	b := UDINT_TO_INT(SIZE) - 1;
	FOR a := 0 TO b DO
		d := d + 1;
		e := e + sbox[d];
		v := sbox[d];
		sbox[d] := sbox[e];
		sbox[e] := v;
		v := sbox[d] + sbox[e];
		BUF[a] :=BUF[a] XOR sbox[v];
	END_FOR;

	POS := POS + SIZE;
	SIZE := MIN(64,end - POS);

	IF SIZE = 0 THEN
		MODE := 3;
	END_IF;
END_CASE;

(* revision history

ks	9. Jan. 2010 rev 1.0
	original version

*)

END_FUNCTION_BLOCK

// POUs/DEMO/SHA1_MD5_DEMO
PROGRAM SHA1_MD5_DEMO
VAR
	text: STRING(OSCAT_BASIC.STRING_LENGTH) := '<4036.1076324381@guildenstern.zeitform.de>';
	MD5_STR : MD5_STR;
	SHA1_STR : SHA1_STR;
	md5_hash : ARRAY [0..15] OF BYTE;
	sha1_hash : ARRAY [0..19] OF BYTE;
	start1 : BOOL := TRUE;
	start2 : BOOL := TRUE;
	done1 : BOOL;
	done2 : BOOL;
	md5_strh : STRING(32);
	sha1_strh : STRING(40);
END_VAR

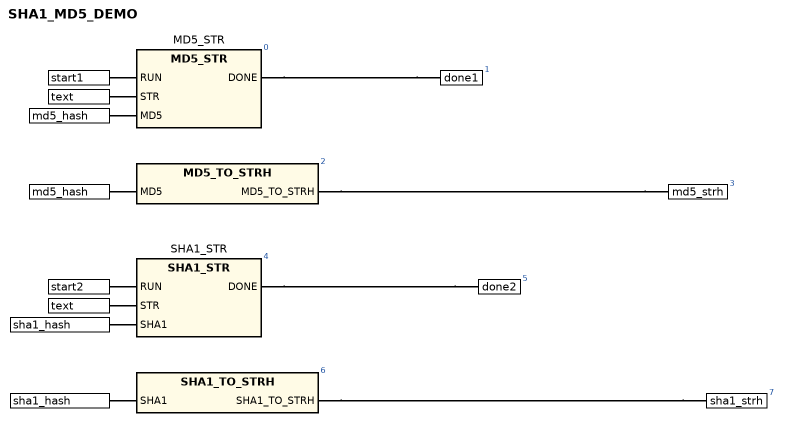
MD5_STR(RUN := start1, STR := text, MD5 := md5_hash);
done1 := MD5_STR.DONE;
md5_strh := MD5_TO_STRH(MD5 := md5_hash);
SHA1_STR(RUN := start2, STR := text, SHA1 := sha1_hash);
done2 := SHA1_STR.DONE;
sha1_strh := SHA1_TO_STRH(SHA1 := sha1_hash);

END_PROGRAM

// POUs/CONVERT/SHA1_STR
FUNCTION_BLOCK SHA1_STR
VAR_INPUT
	RUN: BOOL;
END_VAR
VAR_OUTPUT
	DONE: BOOL;
END_VAR
VAR_IN_OUT
	STR: STRING(OSCAT_BASIC.STRING_LENGTH);
	SHA1 : ARRAY [0..19] OF BYTE;
END_VAR

VAR
	run_last: BOOL;
	SHA1_STREAM : SHA1_STREAM;
	buf : ARRAY [0..63] OF BYTE;
	mode : INT;
	size : UDINT;
	pos : UDINT;
END_VAR

(*
version 1.0	06. dec. 2009
programmer 	ks
tested BY	ks

SHA1_STR berechnet den MD5 Hash eines Strings
*)

CASE mode OF
0:	(* Wait für Start *)
	IF RUN AND NOT run_last THEN
		DONE := FALSE;
		mode := 1; (* Initialisierung *)
		size := LEN(STR);
	END_IF;

2:	(* Data copy and Calc *)
	IF size > 0 THEN
		OSCAT_BASIC._STRING_TO_BUFFER(STR:=MID(STR, UDINT_TO_INT(SIZE), UDINT_TO_INT(POS) + 1), POS:=0, PT:=ADR(buf), SIZE:=SIZEOF(buf));
	END_IF;

3:	DONE := TRUE;
	mode := 0; (* Stop *)

END_CASE;

IF mode > 0 THEN
	SHA1_STREAM(SIZE:=size, MODE:=mode, BUF:=buf, SHA1:=SHA1, POS=>pos);
END_IF;

run_last := RUN;

(* revision history

ks	6. dec. 2009 rev 1.0
	original version

*)

END_FUNCTION_BLOCK

// POUs/CONVERT/SHA1_TO_STRH
FUNCTION SHA1_TO_STRH : STRING(40)
VAR_INPUT
	SHA1 : ARRAY [0..19] OF BYTE;
END_VAR
VAR
	i : INT;
	tmp : BYTE;
	pt : POINTER TO BYTE;
END_VAR
(*
version 1.1	03. dec. 2011
programmer 	ks
tested BY	ks

SHA1_TO_STRH konvertiert das SHA1 Hash Array in einen HEX-String
*)

pt := ADR(SHA1_TO_STRH); (* read output adress to pointer *)

FOR i := 0 TO 19 DO; (* write the 10 hex characters backwards *)
	tmp := SHR(SHA1[i],4);
	PT^ := tmp + SEL(tmp <= 9,87,48);
	pt := pt + 1; (* decrement the pointer *)
	tmp := SHA1[i] AND 2#1111;
	PT^ := tmp + SEL(tmp <= 9,87,48);
	pt := pt + 1; (* decrement the pointer *)
END_FOR;
pt^:= 0; (* write the closing byte for the string *)

(* revision history

ks	6. dec. 2009 rev 1.0
	original version

ks	3. dec. 2011 rev 1.1
	incorrect string size
*)

END_FUNCTION

// POUs/DEMO/SMTP_CLIENT_DEMO
PROGRAM SMTP_CLIENT_DEMO
VAR
(*
	smtp_server: STRING := 'oscat_test%freenet.de:oscat123456@mx.freenet.de';
	smtp_mailfrom: STRING := 'oscat_test@freenet.de';
*)

	SMTP_CLIENT: SMTP_CLIENT;
	smtp_activate: BOOL;
	smtp_timeout: TIME := T#30s;
	smtp_error_t: BYTE;
	smtp_error_c: DWORD;
	smtp_busy: BOOL;
	smtp_done: BOOL;
	smtp_dti: DT;
	smtp_dti_offset: INT := 60;
	smtp_files: STRING(OSCAT_BASIC.STRING_LENGTH) := '';
	smtp_server: STRING := '110876022:oscat123456@mail.gmx.net';
	smtp_mailfrom: STRING := 'oscat@gmx.net;Station_01';
	smtp_mailto: STRING(OSCAT_BASIC.STRING_LENGTH) := 'oscat@gmx.net';
	smtp_subject: STRING := 'Das ist der Betreff';
	smtp_body: STRING(OSCAT_BASIC.STRING_LENGTH) := 'Das ist der Email-Text';
END_VAR
VAR // added by the converter: edge detectors and wires of the graphical bodies
    _w1 : ANY;
END_VAR

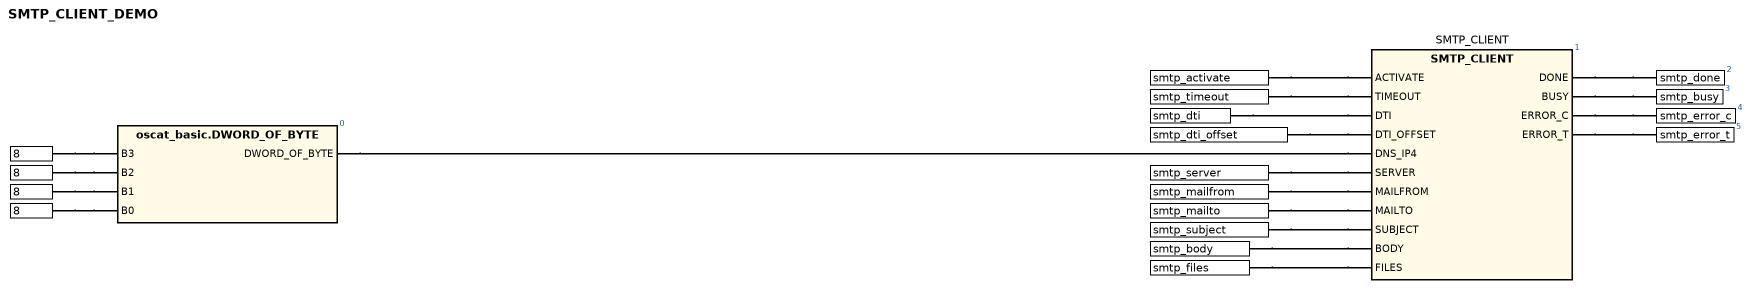
_w1 := oscat_basic.DWORD_OF_BYTE(B3 := 8, B2 := 8, B1 := 8, B0 := 8);
SMTP_CLIENT(
    ACTIVATE := smtp_activate,
    TIMEOUT := smtp_timeout,
    DTI := smtp_dti,
    DTI_OFFSET := smtp_dti_offset,
    DNS_IP4 := _w1,
    SERVER := smtp_server,
    MAILFROM := smtp_mailfrom,
    MAILTO := smtp_mailto,
    SUBJECT := smtp_subject,
    BODY := smtp_body,
    FILES := smtp_files);
smtp_done := SMTP_CLIENT.DONE;
smtp_busy := SMTP_CLIENT.BUSY;
smtp_error_c := SMTP_CLIENT.ERROR_C;
smtp_error_t := SMTP_CLIENT.ERROR_T;

END_PROGRAM

// POUs/NETWORK/SPIDER_ACCESS
FUNCTION_BLOCK SPIDER_ACCESS
VAR_IN_OUT
	IP_C : IP_C;(*IP_Control Verwaltungsstruktur*)
	S_BUF : NETWORK_BUFFER;
	R_BUF : NETWORK_BUFFER;
	VALUE : STRING;
	VAR_NAME : STRING(40);
END_VAR
VAR_INPUT
	MODE : BYTE;
END_VAR
VAR_OUTPUT
	ERROR : DWORD;
END_VAR
VAR
	state : INT;
	st_tmp : STRING(OSCAT_BASIC.STRING_LENGTH);
	URL_DATA : url;
	HTTP_GET : HTTP_GET;
	value_len :	UINT;
	body_len :	UINT;
	mode_save : BYTE;
END_VAR

(*
version 1.1	12. apr. 2011
programmer 	ks
tested by		ks
*)

CASE state OF

00:
	IF MODE > BYTE#0 AND MODE < BYTE#3 THEN
		MODE_SAVE := MODE; (* Modus speichern *)
		(* wenn kein '.' in Name dann ist es eine globale variable *)
		IF FIND(VAR_NAME,'.') = 0 THEN
			st_tmp := CONCAT('%40GV.',VAR_NAME);
		ELSE
			st_tmp := VAR_NAME;
		END_IF;

		IF MODE_SAVE = BYTE#2 THEN (* 2 = Write *)
			VALUE_LEN := INT_TO_UINT(LEN(VALUE));
			st_tmp := CONCAT(st_tmp,'+');
			st_tmp := CONCAT(st_tmp,VALUE);
			URL_DATA:=STRING_TO_URL(STR:= CONCAT('http://x/dir/cgi-bin/writeVal.exe?',st_tmp),DEFAULT_PROTOCOL:='',DEFAULT_PATH:='');
		ELSE
			URL_DATA:=STRING_TO_URL(STR:= CONCAT('http://x/dir/cgi-bin/readVal.exe?',st_tmp),DEFAULT_PROTOCOL:='',DEFAULT_PATH:='');
		END_IF;

		state := 60;
	END_IF;
60:
	IF HTTP_GET.DONE THEN
		IF MODE_SAVE = BYTE#2 THEN (* Write *)
			BODY_LEN := HTTP_GET.BODY_STOP - HTTP_GET.BODY_START + BOOL_TO_UINT(HTTP_GET.BODY_STOP > UINT#0);
			ERROR := BOOL_TO_DWORD(BODY_LEN <> VALUE_LEN);
		ELSE (* Read *)
			IF HTTP_GET.BODY_START > 0 THEN
				VALUE := OSCAT_BASIC.BUFFER_TO_STRING(PT:=ADR(R_BUF.BUFFER),SIZE:=R_BUF.SIZE,START:=UINT_TO_INT(HTTP_GET.BODY_START),STOP:=UINT_TO_INT(HTTP_GET.BODY_STOP));
			ELSE
				VALUE := '';
			END_IF;
		END_IF;
		STATE   := 100;

	ELSIF (HTTP_GET.ERROR > DWORD#00) THEN
		ERROR := HTTP_GET.ERROR;
		STATE   := 100;
	END_IF;

100:
	(* UNLOCK HTTP DATA *)
	IF HTTP_GET.DONE = FALSE THEN
		STATE := 0;
	END_IF;

END_CASE;

(* HTTP_GET *)
HTTP_GET(	IP_C:=IP_C,
			S_BUF:=S_BUF,
			R_BUF:=R_BUF,
			IP4:=DWORD#00,
			GET:=state=60,
			MODE:=BYTE#0,
			UNLOCK_BUF:=state=100,
			URL_DATA:=URL_DATA
			);

(* revision history
ks	18. mar. 2009	rev 1.0
	original version

ks	12. apr. 2011	rev 1.1
	fehlerkorrektur bei buffer_to_string
*)

END_FUNCTION_BLOCK

// POUs/DEMO/SPIDER_DEMO
PROGRAM SPIDER_DEMO
VAR
	SPIDER_ACCESS: SPIDER_ACCESS;
	IP_CONTROL: IP_CONTROL;
	S_BUF: NETWORK_BUFFER;
	R_BUF: NETWORK_BUFFER;
	MODE: BYTE := 1;
	IP_C: IP_C;
	VALUE: STRING;
	VAR_NAME: STRING(40) := 'RTC_SECONDS';
	ERROR: DWORD;
END_VAR
VAR // added by the converter: edge detectors and wires of the graphical bodies
    _w1 : ANY;
END_VAR

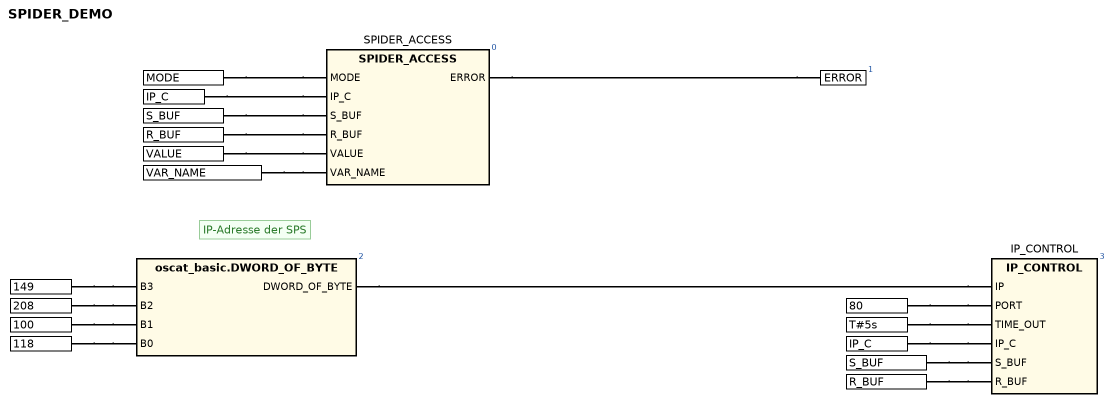
SPIDER_ACCESS(
    MODE := MODE,
    IP_C := IP_C,
    S_BUF := S_BUF,
    R_BUF := R_BUF,
    VALUE := VALUE,
    VAR_NAME := VAR_NAME);
ERROR := SPIDER_ACCESS.ERROR;
// IP-Adresse der SPS
_w1 := oscat_basic.DWORD_OF_BYTE(B3 := 149, B2 := 208, B1 := 100, B0 := 118);
IP_CONTROL(IP := _w1, PORT := 80, TIME_OUT := T#5s, IP_C := IP_C, S_BUF := S_BUF, R_BUF := R_BUF);

END_PROGRAM

// POUs/NETWORK/TELNET_LOG
FUNCTION_BLOCK TELNET_LOG
VAR_IN_OUT
	IP_C : IP_C;
	S_BUF : NETWORK_BUFFER;
	LOG_CL : LOG_CONTROL;
END_VAR
VAR_INPUT
	ENABLE : BOOL;
	OPTION : BYTE := BYTE#2#1000_1100; (* no flush buffer (7) , CR&LF (3), Colors (2), AUTOWRAP (1), Screen-Init (0) *)
	PORT : WORD := 23; (* Port Nummer *)
END_VAR
VAR_OUTPUT
	READY : BOOL;
END_VAR
VAR
	TELNET_PRINT : TELNET_PRINT;
	done : BOOL;
	init : BOOL;
	watchdog : TON;
	ci : INT;
	pi : INT;
	pi_last : INT;
	send : BOOL;
END_VAR

(*
version 1.1	03. Dec. 2011
programmer 	ks
tested BY	ks

TELNET_LOG sendet alle Texte vom LOG_BUFFER an eine TELNET_Konsole
*)

IF NOT init THEN
	init := TRUE;
	IF OPTION > 0 THEN
		TELNET_PRINT.OPTION := OPTION;
	END_IF;
	IF PORT > 0 THEN (* bei portvorgabe wird der standardport überschrieben *)
		TELNET_PRINT.PORT := PORT;
	END_IF;
  	WATCHDOG.PT := T#1ms;
END_IF;

WATCHDOG(IN:=FALSE); (* Timer stoppen *)

ci := LOG_CL.IDX;

(* CONNECT_OFF Flanke auswerten *)
IF IP_C.C_STATE = BYTE#1 THEN
	pi := 0;
	init := FALSE;
END_IF;

REPEAT
	IF pi <> ci AND IP_C.C_STATE > BYTE#127 THEN
		IF pi = 0 AND LOG_CL.RING_MODE THEN pi := ci; END_IF;
		pi_last := pi;
		pi := pi + 1;
		IF pi > LOG_CL.SIZE THEN pi := 1; END_IF;
		SEND := TRUE;
	ELSE
		SEND := FALSE;
	END_IF;

	TELNET_PRINT(	IP_C := IP_C,
					S_BUF := S_BUF,
					ENABLE := ENABLE,
					SEND := SEND,
					TEXT := LOG_CL.MSG[pi],
					BACK_COLOR := DWORD_TO_BYTE(SHL(LOG_CL.MSG_OPTION[pi],8)),
					FRONT_COLOR := DWORD_TO_BYTE(LOG_CL.MSG_OPTION[pi] ));
	READY := TELNET_PRINT.READY;
	done := TELNET_PRINT.DONE;

	IF SEND AND NOT done THEN
		pi := pi_last;
	END_IF;

	WATCHDOG(IN:=TRUE);

UNTIL (WATCHDOG.Q OR NOT done )
END_REPEAT;

(* revision history
ks	14. aug. 2009	rev 1.0
	original version

ks	03. dec. 2011	rev 1.1
	neue parameter und initialisierung optimiert

*)

END_FUNCTION_BLOCK

// POUs/NETWORK/TELNET_PRINT
FUNCTION_BLOCK TELNET_PRINT
VAR_IN_OUT
	IP_C : IP_C;
	S_BUF : NETWORK_BUFFER;
END_VAR
VAR_INPUT
	TEXT : STRING(OSCAT_BASIC.STRING_LENGTH);
	ENABLE : BOOL;
	SEND : BOOL;
	OPTION : BYTE := BYTE#2#1000_1100; (* no flush buffer (7) , CR&LF (3), Colors (2), AUTOWRAP (1), Screen-Init (0) *)
	BACK_COLOR : BYTE;
	FRONT_COLOR : BYTE;
	X_POS : BYTE;
	Y_POS : BYTE;
	PORT : WORD := 23; (* Port Nummer *)
END_VAR
VAR_OUTPUT
	READY : BOOL;
	DONE : BOOL;
END_VAR
VAR
	last_fc : BYTE;
	state : INT;
	x : INT := -1;
	ip_state : BYTE;
	ip_id : BYTE;
	IP_FIFO : IP_FIFO;
	init : BOOL;
	b0_screen_clear : BOOL;
	b1_autowrap : BOOL;
	b2_color : BOOL;
	b3_cr_lr : BOOL;
	b7_no_flush : BOOL;
END_VAR

(*
version 1.4		03. dec. 2011
programmer 		ks
tested by			ks

TELNET_PRINT sendet einem TEXT in Farbe an Position X,Y an eine TELNET-Konsole
*)

READY := IP_C.C_STATE > BYTE#127;
DONE := FALSE;

CASE state OF

00: (* Warten auf Freigabe *)
	IF ENABLE THEN
		state := 10;
		ip_state := BYTE#1; (* Anmelden *)
	END_IF;

10: (* Bei IP_Control anmelden und auf freigabe warten *)
	IF ip_state = BYTE#3 THEN

		(* IP Datenverkehr einrichten *)
		IP_C.C_PORT := PORT; (* Portnummer eintragen *)
		IP_C.C_IP := DWORD#00; (* IP eintragen *)
		IP_C.C_MODE := BYTE#4; (* Mode: TCP+PASSIV+PORT *)
		IP_C.TIME_RESET := TRUE; (* Zeitueberwachung rücksetzen *)
		IP_C.C_ENABLE := TRUE; (* Verbindungsaufbau freigeben *)
		IP_C.R_OBSERVE := FALSE; (* keine Empfangsueberwachung *)
		state := 20;
	END_IF;

20:	IF IP_C.ERROR > DWORD#0 THEN
		IP_C.TIME_RESET := TRUE; (* Fehler rücksetzen *)
	END_IF;
	IF S_BUF.SIZE = UINT#0 THEN (* Datensenden nicht aktiv *)
		IF NOT ENABLE THEN
			ip_state := BYTE#4; (* Verbindung abbauen - Ressource freigeben *)
			IP_C.C_ENABLE := FALSE; (* Verbindungsabbau *)
			state := 0;
		END_IF;
		IF IP_C.C_STATE = BYTE#1 THEN (* positive Flanke Connect off *)
			init := FALSE;
		ELSIF READY THEN (* Verbindung vorhanden *)
			IF IP_C.C_STATE = BYTE#254 AND NOT INIT THEN (* positive Flanke Connect on *)
				(* Var Init ist notwendig, damit der Baustein im selben zyklus mehrmals ausgerufen werden kann *)
				init := TRUE;
				b0_screen_clear := (OPTION AND BYTE#2#0000_0001) > BYTE#0;
				b1_autowrap := (OPTION AND BYTE#2#0000_0010) > BYTE#0;
				b2_color := (OPTION AND BYTE#2#0000_0100) > BYTE#0;
				b3_cr_lr := (OPTION AND BYTE#2#0000_1000) > BYTE#0;
				b7_no_flush := (OPTION AND BYTE#2#1000_0000) > BYTE#0;

				last_fc := NOT FRONT_COLOR; (* aktualisierung der Farben erzwingen !*)
				x := 0;

				(* AUTOWRAP OFF/ON *)
				S_BUF.BUFFER[x] := BYTE#16#1B; (* ESC *)
				x := x +1;
				S_BUF.BUFFER[x] := BYTE#16#5B; (* [ *)
				x := x +1;
				S_BUF.BUFFER[x] := BYTE#16#3F; (* ? *)
				x := x +1;
				S_BUF.BUFFER[x] := BYTE#16#37; (* 7 *)
				x := x +1;
				S_BUF.BUFFER[x] := SEL(b1_autowrap, BYTE#16#6C (* l *),BYTE#16#68 (* h *));

				IF b0_screen_clear THEN
					IF b2_color THEN
						x := x +1;
						S_BUF.BUFFER[x] := BYTE#16#1B; (* ESC *)
						x := x +1;
						S_BUF.BUFFER[x] := BYTE#16#5B; (* [ *)
						x := x +1;
						S_BUF.BUFFER[x] := BYTE#16#30; (* 0 *)
						x := x +1;
						S_BUF.BUFFER[x] := BYTE#16#3B; (* ; *)
						x := x +1;
						S_BUF.BUFFER[x] := BYTE#16#33; (* 3 *)
						x := x +1;
						S_BUF.BUFFER[x] := (FRONT_COLOR AND BYTE#2#00000111) OR BYTE#16#30; (* Einerstelle Farbe Foreground ausgeben *)
						x := x +1;
						S_BUF.BUFFER[x] := BYTE#16#3B; (* ; *)
						x := x +1;
						S_BUF.BUFFER[x] := BYTE#16#34; (* 4 *)
						x := x +1;
						S_BUF.BUFFER[x] := (BACK_COLOR AND BYTE#2#00000111) OR BYTE#16#30; (* Einerstelle Farbe Background ausgeben *)
						x := x +1;
						S_BUF.BUFFER[x] := BYTE#16#6D; (* m *)
					END_IF;
					(* Screen Clear *)
					x := x +1;
					S_BUF.BUFFER[x] := BYTE#16#1B; (* ESC *)
					x := x +1;
					S_BUF.BUFFER[x] := BYTE#16#5B; (* [ *)
					x := x +1;
					S_BUF.BUFFER[x] := BYTE#16#32; (* 2 *)
					x := x +1;
					S_BUF.BUFFER[x] := BYTE#16#4A; (* J *)
				ELSE
					x := x +1;
					S_BUF.BUFFER[x] := BYTE#16#0A; (* neue Zeile *)
				END_IF;
			END_IF;

			(* buffer voll , oder Daten sind vorhanden und kein weiterer Sendewunsch *)
			IF (INT_TO_UINT(x + LEN(TEXT) + 21) > SIZEOF(S_BUF.BUFFER)) OR (x >= 0 AND NOT SEND) THEN
				S_BUF.SIZE := INT_TO_UINT(x + 1); (* Länge eintragen -> Datensenden starten *)
				x := -1;
			ELSIF SEND THEN

				(* aktuelle Farbe bestimmen  *)
				IF b2_color AND FRONT_COLOR <> last_FC THEN
					(* Farbeinstellung: ANSI-Sequenz ESC[X;Y;Zm ausgeben *)
					x := x + 1;
					S_BUF.BUFFER[x] := BYTE#16#1B; (* ESC *)
					x := x + 1;
					S_BUF.BUFFER[x] := BYTE#16#5B; (* [ *)
					(* Farbeinstellung: dunkel oder Hell und blinken bestimmen *)
					IF ((FRONT_COLOR AND BYTE#2#0001_1000) XOR (last_FC AND BYTE#2#0001_1000)) <> BYTE#00 OR TRUE THEN
						x := x + 1;
						S_BUF.BUFFER[x] := BYTE#16#30; (* 0  *)
						x := x + 1;
						S_BUF.BUFFER[x] := BYTE#16#3B; (* ; *)
						(* keine dunklen Farben gewünscht -> dann Bold & Bright *)
						IF (FRONT_COLOR AND BYTE#2#00001000) = BYTE#0 THEN
							(* auf Bold & Bright Farben umstellen *)
							x := x + 1;
							S_BUF.BUFFER[x] := BYTE#16#31; (* 1 *)
							x := x + 1;
							S_BUF.BUFFER[x] := BYTE#16#3B; (* ; *)
						END_IF;
						(* blinkenden Farben gewünscht *)
						IF (FRONT_COLOR AND BYTE#2#00010000) > BYTE#0 THEN
							(* auf Blinkenden Farbe umstellen *)
							x := x + 1;
							S_BUF.BUFFER[x] := BYTE#16#35; (* 5 *)
							x := x + 1;
							S_BUF.BUFFER[x] := BYTE#16#3B; (* ; *)
						END_IF;
					END_IF;
					(* Zehnerstelle Farbe Foreground ausgeben *)
					x := x + 1;
					S_BUF.BUFFER[x] := BYTE#16#33; (* 3 *)
					(* Einerstelle Farbe Foreground ausgeben *)
					x := x + 1;
					S_BUF.BUFFER[x] := (FRONT_COLOR AND BYTE#2#00000111) OR BYTE#16#30;
					x := x + 1;
					S_BUF.BUFFER[x] := BYTE#16#6D; (* m *)
					(* neue Farbe als letzt verwendete speichern *)
					last_FC := FRONT_COLOR;
				END_IF;

				(* Cursor positionieren *)
				IF X_POS > BYTE#0 AND Y_POS > BYTE#0 THEN
					x := x + 1;
					S_BUF.BUFFER[x] := BYTE#16#1B; (* ESC *)
					x := x + 1;
					S_BUF.BUFFER[x] := BYTE#16#5B; (* [ *)
					(* Zehnerstelle Y_POS ausgeben *)
					x := x + 1;
					S_BUF.BUFFER[x] := SHR(OSCAT_BASIC.INT_TO_BCDC(BYTE_TO_INT(Y_POS)),4) OR BYTE#16#30;
					(* Einerstelle Y_POS ausgeben *)
					x := x + 1;
					S_BUF.BUFFER[x] := (OSCAT_BASIC.INT_TO_BCDC(BYTE_TO_INT(Y_POS)) AND BYTE#16#0F) OR BYTE#16#30;
					x := x + 1;
					S_BUF.BUFFER[x] := BYTE#16#3B; (* ; *)
					(* Zehnerstelle X_POS ausgeben *)
					x := x + 1;
					S_BUF.BUFFER[x] := SHR(OSCAT_BASIC.INT_TO_BCDC(BYTE_TO_INT(X_POS)),4) OR BYTE#16#30;
					(* Einerstelle X_POS ausgeben *)
					x := x + 1;
					S_BUF.BUFFER[x] := (OSCAT_BASIC.INT_TO_BCDC(BYTE_TO_INT(X_POS)) AND BYTE#16#0F) OR BYTE#16#30;
					x := x + 1;
					S_BUF.BUFFER[x] := BYTE#16#48; (* H *)
				END_IF;

				(* text ausgeben *)
				IF LEN(TEXT) > 0 THEN
					OSCAT_BASIC._STRING_TO_BUFFER(str:=TEXT,pos:=x + 1,pt :=ADR(S_BUF.BUFFER), size:=SIZEOF(S_BUF.BUFFER));
					x := x + LEN(TEXT);
				END_IF;

				IF b3_cr_lr THEN (* Option: CR,LF ausgeben *)
					x := x + 1;
					S_BUF.BUFFER[x] := BYTE#16#0D;
					x := x + 1;
					S_BUF.BUFFER[x] := BYTE#16#0A;
				END_IF;

				DONE := TRUE; (* Fertig in Buffer eingetragen *)

				IF b7_no_flush THEN (* Option: no buffer flush *)
					(* buffer sofort senden - aktuellen Schreibindex speichern -> Senden anstossen *)
					S_BUF.SIZE := INT_TO_UINT(x + 1);
					x := -1;
				END_IF;
			END_IF;
		END_IF;
	END_IF;
END_CASE;

(* IP_FIFO *)
IP_FIFO(FIFO:=IP_C.FIFO,STATE:=ip_state,ID:=ip_id);

(* revision history
ks	05. jan. 2009	rev 1.0
	original version

ks	20. oct. 2009	rev 1.1
	Networkbuffer und Buffer-funktionen auf Basis 0

ks	20. oct. 2009	rev 1.2
	STRING(OSCAT_BASIC.STRING_LENGTH)

ks	17. may. 2011	rev 1.3
	automatischer re-connect

ks	03. dec. 2011	rev 1.4
	initialisierung verbessert, Port Nummer als Parmeter

*)

END_FUNCTION_BLOCK

// POUs/DEMO/TELNET_LOG_DEMO
PROGRAM TELNET_LOG_DEMO
VAR
	TELNET_LOG: TELNET_LOG;
	IPC: IP_C;
	S_BUF: NETWORK_BUFFER;
	R_BUF: NETWORK_BUFFER;
	READY: BOOL;
	IP_CONTROL: IP_CONTROL;
	TON_1: TON;
	LOG_MSG: LOG_MSG;
END_VAR

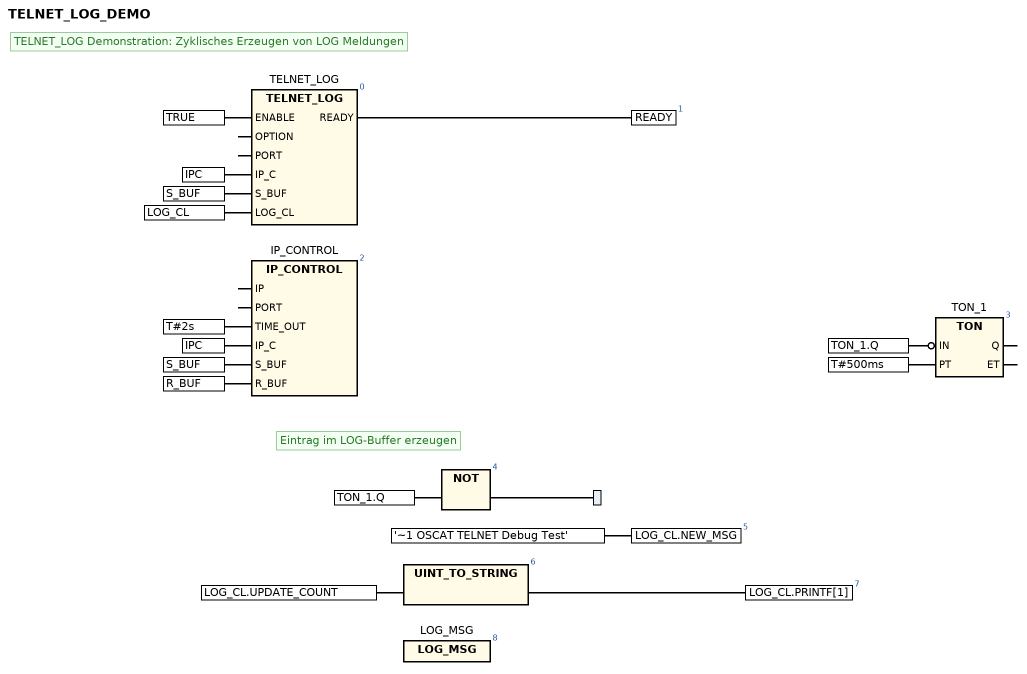
// TELNET_LOG Demonstration: Zyklisches Erzeugen von LOG Meldungen
TELNET_LOG(ENABLE := TRUE, IP_C := IPC, S_BUF := S_BUF, LOG_CL := LOG_CL);
READY := TELNET_LOG.READY;
IP_CONTROL(TIME_OUT := T#2s, IP_C := IPC, S_BUF := S_BUF, R_BUF := R_BUF);
TON_1(IN := NOT TON_1.Q, PT := T#500ms); // TON
// Eintrag im LOG-Buffer erzeugen
(* NOT TON_1.Q; result not used *)
LOG_CL.NEW_MSG := '~1 OSCAT TELNET Debug Test';
LOG_CL.PRINTF[1] := UINT_TO_STRING(LOG_CL.UPDATE_COUNT);
LOG_MSG();

END_PROGRAM

// POUs/DEMO/TELNET_PRINT_DEMO
PROGRAM TELNET_PRINT_DEMO
VAR
	COUNT_BR_1: OSCAT_BASIC.COUNT_BR;
	READY: BOOL;
	TON_1: TON;
	TEXT: STRING;
	TEXT_ATTRIBUTE: BYTE;
	GEN_SIN_1: oscat_basic.GEN_SIN;
	X_POS: BYTE;
	Y_POS: BYTE;
	GEN_SIN_2: oscat_basic.GEN_SIN;
	TELNET_PRINT: TELNET_PRINT;
	DONE: BOOL;
	IP_C: IP_C;
	S_BUF: NETWORK_BUFFER;
	IP_CONTROL: IP_CONTROL;
	R_BUF: NETWORK_BUFFER;
END_VAR
VAR // added by the converter: edge detectors and wires of the graphical bodies
    _w1, _w2 : ANY;
END_VAR

TON_1(IN := NOT TON_1.Q, PT := T#100ms); // TON
COUNT_BR_1(IN := BYTE#1, UP := TON_1.Q AND READY, MX := BYTE#31); // oscat_basic.COUNT_BR
TEXT_ATTRIBUTE := COUNT_BR_1.CNT;
GEN_SIN_1(PT := T#5s, AM := 43.0, OS := 22.0); // oscat_basic.GEN_SIN
_w1 := oscat_basic.STAIR(X := GEN_SIN_1.Out, D := 0.0);
X_POS := REAL_TO_BYTE(_w1);
GEN_SIN_2(PT := T#7s, AM := 24.0, OS := 13.0); // oscat_basic.GEN_SIN
_w2 := oscat_basic.STAIR(X := GEN_SIN_2.Out, D := 0.0);
Y_POS := REAL_TO_BYTE(_w2);
TEXT := CONCAT(STR1 := ' OSCAT TELNET_Print - Test: Color: ', STR2 := BYTE_TO_STRING(TEXT_ATTRIBUTE));
TELNET_PRINT(
    TEXT := TEXT,
    ENABLE := TRUE,
    SEND := TON_1.Q,
    OPTION := BYTE#2#0000_0101,
    BACK_COLOR := BYTE#00,
    FRONT_COLOR := TEXT_ATTRIBUTE,
    X_POS := X_POS,
    Y_POS := Y_POS,
    IP_C := IP_C,
    S_BUF := S_BUF);
READY := TELNET_PRINT.READY;
DONE := TELNET_PRINT.DONE;
IP_CONTROL(TIME_OUT := T#2s, IP_C := IP_C, S_BUF := S_BUF, R_BUF := R_BUF);

END_PROGRAM

// POUs/TELNET_VISION/TN_FRAMEWORK
FUNCTION_BLOCK TN_FRAMEWORK
VAR
	FB_IP_CONTROL : IP_CONTROL;
	FB_TN_INPUT_CONTROL : TN_INPUT_CONTROL;
	FB_TN_INPUT_MENU_BAR : TN_INPUT_MENU_BAR;
	FB_TN_RECEIVE :	TN_RECEIVE;
	FB_TN_SEND_ROWS : TN_SEND_ROWS;
	t : TON;
END_VAR
VAR_IN_OUT
	us_TN_INPUT_CONTROL : us_TN_INPUT_CONTROL;
	us_TN_SCREEN : us_TN_SCREEN;
	us_TN_MENU : us_TN_MENU;
	S_BUF : NETWORK_BUFFER;
	R_BUF : NETWORK_BUFFER;
	IP_C : IP_C;
END_VAR
VAR_INPUT
	PORT : WORD;
END_VAR

(*
version 1.1		17. may 2011
programmer		ks
tested by			ks

TN_FRAMEWORK ist ein Grundgerüst zur Nutzung des TELNET VISION Systems, und beinhält alle Laufzeit Komponenten.
*)

(* Initialisierung / Freigeben der Verbindung *)
IF (NOT IP_C.C_ENABLE) THEN

	(* IP Datenverkehr einrichten *)
	IP_C.C_PORT := SEL(PORT=BYTE#0,PORT,WORD#23); (* Portnummer eintragen *)
	IP_C.C_IP := DWORD#00; (* IP eintragen *)
	IP_C.C_MODE := BYTE#4; (* Mode: TCP+PASSIV+PORT *)
	IP_C.TIME_RESET := TRUE; (* Zeitueberwachung rücksetzen *)
	IP_C.C_ENABLE := TRUE; (* Verbindungsaufbau freigeben *)
	IP_C.R_OBSERVE := FALSE; (* keine Empfangsueberwachung *)

END_IF;

t(IN:= IP_C.ERROR > DWORD#0, PT:=T#5s);
IF t.Q THEN
	IP_C.TIME_RESET := TRUE; (* Error Reset *)
END_IF;

(* Telnet-Menu-Bar *)
FB_TN_INPUT_MENU_BAR(
	Xus_TN_MENU := us_TN_MENU,
	Xus_TN_SCREEN := us_TN_SCREEN);

(* Telnet-Input-Control *)
FB_TN_INPUT_CONTROL(
	Xus_TN_SCREEN := us_TN_SCREEN,
	Xus_TN_INPUT_CONTROL := us_TN_INPUT_CONTROL);

(* Telnet-Data-Send Line-Updates *)
FB_TN_SEND_ROWS(
	IP_C :=IP_C,
	S_BUF :=S_BUF,
	Xus_TN_SCREEN :=us_TN_SCREEN,
	S_BUF_SIZE :=SIZEOF(S_BUF.BUFFER));

(* Telnet-Server *)
FB_IP_CONTROL(
	IP_C :=IP_C,
	S_BUF :=S_BUF,
	R_BUF :=R_BUF,
	IP :=DWORD#00,
	PORT :=WORD#00,
	TIME_OUT :=T#2s);

(* Telnet-Data-Receive *)
FB_TN_RECEIVE(
	R_BUF := R_BUF,
	Xus_TN_SCREEN := us_TN_SCREEN);

(* revision history
ks	10. mai. 2010	rev 1.0
	original version

ks	17. may. 2011	rev 1.1
	automatischer re-connect

ks	05. may. 2012	rev 1.2
	neue parameter PORT
*)

END_FUNCTION_BLOCK

// POUs/TELNET_VISION/TN_INPUT_CONTROL
FUNCTION_BLOCK TN_INPUT_CONTROL
VAR_IN_OUT
	Xus_TN_SCREEN : us_TN_SCREEN;
	Xus_TN_INPUT_CONTROL : us_TN_INPUT_CONTROL;
END_VAR
VAR
	FB_TN_INPUT_SELECT_POPUP : TN_INPUT_SELECT_POPUP;
	FB_TN_INPUT_SELECT_TEXT : TN_INPUT_SELECT_TEXT;
	FB_TN_SC_WRITE_C : TN_SC_WRITE_C;
	FB_TN_INPUT_EDIT_LINE : TN_INPUT_EDIT_LINE;
END_VAR
VAR
	in_index : INT;
	in_Scroll_Offset : INT;
	in_Focus_new : INT;
	in_Focus_alt : INT;
	bo_Tool_Tip_Update : BOOL;
END_VAR

(*
version 1.0		10. mai 2010
programmer		ks
tested by		ks

TN_INPUT_CONTROL dient zur verwaltung und grafischen Darstellung der INPUT_CONTROL Elemente
*)

(* Bearbeitung freigegeben ? *)
IF (Xus_TN_INPUT_CONTROL.bo_Enable = FALSE) OR (Xus_TN_SCREEN.bo_Menue_Bar_Dialog = TRUE) THEN
	RETURN;
END_IF;

(* Fokus Reset durchführen *)
IF (Xus_TN_INPUT_CONTROL.bo_Reset_Fokus = TRUE) THEN
	Xus_TN_INPUT_CONTROL.bo_Reset_Fokus := FALSE;

	FOR in_index := INT#01 TO Xus_TN_INPUT_CONTROL.in_Count DO
		Xus_TN_INPUT_CONTROL.usa_TN_INPUT_CONTROL_DATA[in_index].bo_Focus := FALSE;
	END_FOR;

	IF (Xus_TN_INPUT_CONTROL.in_Count >= INT#01) THEN
		Xus_TN_INPUT_CONTROL.usa_TN_INPUT_CONTROL_DATA[1].bo_Focus := TRUE;
		Xus_TN_INPUT_CONTROL.in_Focus_at := INT#01;
	END_IF;

	Xus_TN_INPUT_CONTROL.bo_Update_all := TRUE;
END_IF;

IF (Xus_TN_SCREEN.bo_Modal_Dialog = FALSE) THEN
	(* TAB-Taste für Control-element wechsel auswerten *)
	IF (Xus_TN_SCREEN.by_Input_Exten_Code = BYTE#09) THEN

		in_Scroll_Offset := INT#01;

		(* Cursor-Oben Taste *)
	ELSIF (Xus_TN_SCREEN.by_Input_Exten_Code = BYTE#65) THEN

		in_Scroll_Offset := -1;

		(* Cursor-unten Taste *)
	ELSIF (Xus_TN_SCREEN.by_Input_Exten_Code = BYTE#66) THEN

		in_Scroll_Offset := INT#01;

	END_IF;
END_IF;

IF (in_Scroll_Offset <> INT#00) THEN  
	(* Grenzwerte überprüfen                                            *)

	Xus_TN_INPUT_CONTROL.in_Focus_at:=LIMIT(INT#01,Xus_TN_INPUT_CONTROL.in_Focus_at,Xus_TN_INPUT_CONTROL.in_Count);

	in_Focus_new := Xus_TN_INPUT_CONTROL.in_Focus_at + in_Scroll_Offset;

	IF (in_Focus_new > Xus_TN_INPUT_CONTROL.in_Count) THEN
		in_Focus_new := INT#1;
	END_IF;

	IF (in_Focus_new < INT#01) THEN
		in_Focus_new := Xus_TN_INPUT_CONTROL.in_Count;
	END_IF;

	in_Focus_alt := Xus_TN_INPUT_CONTROL.in_Focus_at;

	(* aktuellen Element den Fokus entziehen *)
	Xus_TN_INPUT_CONTROL.usa_TN_INPUT_CONTROL_DATA[in_Focus_alt].bo_Focus := FALSE;
	Xus_TN_INPUT_CONTROL.usa_TN_INPUT_CONTROL_DATA[in_Focus_alt].bo_Update_Input := TRUE;

	(* neuem Element den Fokus geben *)
	Xus_TN_INPUT_CONTROL.usa_TN_INPUT_CONTROL_DATA[in_Focus_new].bo_Focus  := TRUE;
	Xus_TN_INPUT_CONTROL.usa_TN_INPUT_CONTROL_DATA[in_Focus_new].bo_Update_Input := TRUE;

	Xus_TN_INPUT_CONTROL.in_Focus_at := in_Focus_new;

	bo_Tool_Tip_Update := TRUE;
	in_Scroll_Offset := INT#00;

END_IF;

(* Alle Elemente updaten ? *)
IF (Xus_TN_INPUT_CONTROL.bo_Update_all = TRUE) THEN
	FOR in_index := 1 TO Xus_TN_INPUT_CONTROL.in_Count DO
		Xus_TN_INPUT_CONTROL.usa_TN_INPUT_CONTROL_DATA[in_index].bo_Update_All := TRUE;
	END_FOR;
	Xus_TN_INPUT_CONTROL.bo_Update_all := FALSE;
	bo_Tool_Tip_Update := TRUE;
END_IF;

FOR in_index := 1 TO Xus_TN_INPUT_CONTROL.in_Count DO

	IF (Xus_TN_INPUT_CONTROL.usa_TN_INPUT_CONTROL_DATA[in_index].in_Type > INT#00) THEN

		IF (Xus_TN_INPUT_CONTROL.usa_TN_INPUT_CONTROL_DATA[in_index].bo_Focus = TRUE) THEN

			Xus_TN_INPUT_CONTROL.usa_TN_INPUT_CONTROL_DATA[in_index].by_Input_ASCII_Code  := Xus_TN_SCREEN.by_Input_ASCII_Code;
			Xus_TN_INPUT_CONTROL.usa_TN_INPUT_CONTROL_DATA[in_index].by_Input_Exten_Code  := Xus_TN_SCREEN.by_Input_Exten_Code;
			Xus_TN_INPUT_CONTROL.usa_TN_INPUT_CONTROL_DATA[in_index].bo_Input_ASCII_IsNum := Xus_TN_SCREEN.bo_Input_ASCII_IsNum;

			(* Tool-Tip Text ausgeben *)
			IF (bo_Tool_Tip_Update = TRUE) THEN

				FB_TN_SC_WRITE_C(	Iin_Y := Xus_TN_INPUT_CONTROL.in_ToolTip_Y,
									Iin_X := Xus_TN_INPUT_CONTROL.in_ToolTip_X,
									Iby_ATTR := Xus_TN_INPUT_CONTROL.by_ToolTip_Attr,
									Iin_OPTION := INT#02, (* Center-String *)
									Iin_LENGTH := Xus_TN_INPUT_CONTROL.in_ToolTip_Size,
									Ist_STRING := Xus_TN_INPUT_CONTROL.usa_TN_INPUT_CONTROL_DATA[in_index].st_Input_ToolTip,
									Xus_TN_SCREEN := Xus_TN_SCREEN);

				(* Flag rücksetzen *)
				bo_Tool_Tip_Update := FALSE;
			END_IF;
		END_IF;

		CASE Xus_TN_INPUT_CONTROL.usa_TN_INPUT_CONTROL_DATA[in_index].in_Type OF
		1:
			(* Edit-Line bearbeiten *)
			FB_TN_INPUT_EDIT_LINE(	Xus_TN_INPUT_CONTROL_DATA := Xus_TN_INPUT_CONTROL.usa_TN_INPUT_CONTROL_DATA[in_index],
									Xus_TN_SCREEN := Xus_TN_SCREEN);
		2:
			(* Select-Text bearbeiten *)
			FB_TN_INPUT_SELECT_TEXT(	Xus_TN_INPUT_CONTROL_DATA := Xus_TN_INPUT_CONTROL.usa_TN_INPUT_CONTROL_DATA[in_index],
										Xus_TN_SCREEN := Xus_TN_SCREEN);
		3:
			(* Select-Popup bearbeiten *)
			FB_TN_INPUT_SELECT_POPUP(	Xus_TN_INPUT_CONTROL_DATA := Xus_TN_INPUT_CONTROL.usa_TN_INPUT_CONTROL_DATA[in_index],
										Xus_TN_SCREEN := Xus_TN_SCREEN);
		END_CASE;

		IF (Xus_TN_INPUT_CONTROL.usa_TN_INPUT_CONTROL_DATA[in_index].bo_Focus = TRUE) THEN

			(* Cursor position von Element auf Screen übertragen *)
			Xus_TN_SCREEN.in_Cursor_X := Xus_TN_INPUT_CONTROL.usa_TN_INPUT_CONTROL_DATA[in_index].in_Cursor_X;
			Xus_TN_SCREEN.in_Cursor_Y := Xus_TN_INPUT_CONTROL.usa_TN_INPUT_CONTROL_DATA[in_index].in_Cursor_Y;

		END_IF;
	END_IF;
END_FOR;

(* revision history
ks	10. mai. 2010	rev 1.0
	original version
*)

END_FUNCTION_BLOCK

// POUs/TELNET_VISION/TN_INPUT_SELECT_POPUP
FUNCTION_BLOCK TN_INPUT_SELECT_POPUP
VAR
	in_index : INT;
	in_Element_Count : INT;
	by_Cur_Key : BYTE;
	by_Attr : BYTE;
	st_String : STRING;
END_VAR
VAR
	us_TN_MENU_POPUP : us_TN_MENU_POPUP;
	FB_TN_INPUT_MENU_POPUP : TN_INPUT_MENU_POPUP;
	FB_TN_SC_WRITE : TN_SC_WRITE;
END_VAR
VAR_IN_OUT
	Xus_TN_SCREEN : us_TN_SCREEN;
	Xus_TN_INPUT_CONTROL_DATA : us_TN_INPUT_CONTROL_DATA;
END_VAR

(*
version 1.1		06. apr 2011
programmer		ks
tested by			ks

TN_SELECT_POPUP dient zur verwaltung und darstellung eines POPUP-Dialogs zur Elementeauswahl
*)

(* Benutzereingabe auswerten -> Selektion Text n *)
IF (Xus_TN_INPUT_CONTROL_DATA.bo_Focus = TRUE) THEN

	by_Cur_Key := Xus_TN_INPUT_CONTROL_DATA.by_Input_Exten_Code;

	IF (us_TN_MENU_POPUP.bo_Activ = FALSE) THEN
		us_TN_MENU_POPUP.by_Input_Exten_Code := BYTE#00;

		(* Return-Taste auswerten *)
		IF (by_Cur_Key = BYTE#13) THEN
			(* Popup-Menu parameter übergeben *)
			us_TN_MENU_POPUP.in_Y := Xus_TN_INPUT_CONTROL_DATA.in_Y;
			us_TN_MENU_POPUP.in_X := Xus_TN_INPUT_CONTROL_DATA.in_X;
			us_TN_MENU_POPUP.by_Attr_mF := Xus_TN_INPUT_CONTROL_DATA.by_Attr_mF;
			us_TN_MENU_POPUP.by_Attr_oF := Xus_TN_INPUT_CONTROL_DATA.by_Attr_oF;
			us_TN_MENU_POPUP.st_Menu_Text := Xus_TN_INPUT_CONTROL_DATA.st_Input_Data;
			us_TN_MENU_POPUP.bo_Create := TRUE;
			us_TN_MENU_POPUP.in_Cur_Item := INT#00;
		END_IF;

		IF (us_TN_MENU_POPUP.in_Cur_Item > INT#00) THEN
			Xus_TN_INPUT_CONTROL_DATA.in_selected := us_TN_MENU_POPUP.in_Cur_Item;
			Xus_TN_INPUT_CONTROL_DATA.bo_Input_Entered := TRUE;
			Xus_TN_INPUT_CONTROL_DATA.bo_Update_Input := TRUE;
			us_TN_MENU_POPUP.in_Cur_Item := INT#00;
		END_IF;

	ELSE
		us_TN_MENU_POPUP.by_Input_Exten_Code := by_Cur_Key;
	END_IF;

	(* Popup-Menu zyklisch aufrufen *)
	FB_TN_INPUT_MENU_POPUP(Xus_TN_MENU_POPUP := us_TN_MENU_POPUP, Xus_TN_SCREEN := Xus_TN_SCREEN);

END_IF;

(* Aktualisierung der Anzeige *)
IF (Xus_TN_INPUT_CONTROL_DATA.bo_Update_Input = TRUE) OR (Xus_TN_INPUT_CONTROL_DATA.bo_Update_All = TRUE) THEN

	(* Title-Text ausgeben *)
	IF Xus_TN_INPUT_CONTROL_DATA.bo_Update_All = TRUE THEN

		IF (Xus_TN_INPUT_CONTROL_DATA.in_Title_X_Offset = INT#00) AND (Xus_TN_INPUT_CONTROL_DATA.in_Title_Y_Offset = INT#00) THEN
			(* wenn Offset X,Y =0 dann Titlestring links vom Element positionieren *)
			FB_TN_SC_WRITE.Iin_Y := Xus_TN_INPUT_CONTROL_DATA.in_Y;
			FB_TN_SC_WRITE.Iin_X := Xus_TN_INPUT_CONTROL_DATA.in_X - LEN(Xus_TN_INPUT_CONTROL_DATA.st_Title_String);

		ELSE
			(* Title-Text durch Row, Color-Offset ausgeben *)
			FB_TN_SC_WRITE.Iin_Y := Xus_TN_INPUT_CONTROL_DATA.in_Y + Xus_TN_INPUT_CONTROL_DATA.in_Title_Y_Offset;
			FB_TN_SC_WRITE.Iin_X := Xus_TN_INPUT_CONTROL_DATA.in_X + Xus_TN_INPUT_CONTROL_DATA.in_Title_X_Offset;
		END_IF;

		(* Title-Text durch Row, Color-Offset ausgeben *)
		FB_TN_SC_WRITE(	Iby_ATTR := Xus_TN_INPUT_CONTROL_DATA.by_Title_Attr,
						Ist_STRING := Xus_TN_INPUT_CONTROL_DATA.st_Title_String,
						Xus_TN_SCREEN := Xus_TN_SCREEN);
	END_IF;

	in_Element_Count := ELEMENT_COUNT(SEP:=BYTE#35,ELEMENT:=Xus_TN_INPUT_CONTROL_DATA.st_Input_Data);

	IF in_Element_Count > INT#00 THEN

		Xus_TN_INPUT_CONTROL_DATA.in_selected:=LIMIT(1,Xus_TN_INPUT_CONTROL_DATA.in_selected,in_Element_Count);

		in_index := Xus_TN_INPUT_CONTROL_DATA.in_selected;

		st_String := ELEMENT_GET(SEP:=BYTE#35,POS:=in_index - 1,ELEMENT:=Xus_TN_INPUT_CONTROL_DATA.st_Input_Data);

		st_String:= OSCAT_BASIC.FIX(str:=st_String,
						L:=LEN(Xus_TN_INPUT_CONTROL_DATA.st_Input_Mask),
						C:=BYTE#32,
						M:=Xus_TN_INPUT_CONTROL_DATA.in_Input_Option);


		Xus_TN_INPUT_CONTROL_DATA.st_Input_String := st_String;

		IF Xus_TN_INPUT_CONTROL_DATA.bo_Focus = TRUE THEN
			by_Attr := Xus_TN_INPUT_CONTROL_DATA.by_Attr_mF;
		ELSE
			by_Attr := Xus_TN_INPUT_CONTROL_DATA.by_Attr_oF;
		END_IF;

		FB_TN_SC_WRITE(	Iin_X := Xus_TN_INPUT_CONTROL_DATA.in_X,
								Iin_Y := Xus_TN_INPUT_CONTROL_DATA.in_Y,
								Iby_ATTR := by_Attr,
								Ist_STRING := st_String,
								Xus_TN_SCREEN := Xus_TN_SCREEN );
	END_IF;

	(* Cursor auf aktuelle Position setzen *)
	Xus_TN_INPUT_CONTROL_DATA.in_Cursor_X := Xus_TN_INPUT_CONTROL_DATA.in_X;
	Xus_TN_INPUT_CONTROL_DATA.in_Cursor_Y := Xus_TN_INPUT_CONTROL_DATA.in_Y;

	(* Update-Flag's rücksetzen *)
	Xus_TN_INPUT_CONTROL_DATA.bo_Update_All   := FALSE;
	Xus_TN_INPUT_CONTROL_DATA.bo_Update_Input := FALSE;

END_IF;

(* revision history

ks	06. apr. 2011	rev 1.1
	list_len und list_get durch element_count und element_get ersetzt

ks	10. mai. 2010	rev 1.0
	original version
*)

END_FUNCTION_BLOCK

// POUs/TELNET_VISION/TN_INPUT_MENU_POPUP
FUNCTION_BLOCK TN_INPUT_MENU_POPUP
VAR
	FB_TN_SC_AREA_SAVE : TN_SC_AREA_SAVE;
	FB_TN_SC_AREA_RESTORE : TN_SC_AREA_RESTORE;
	FB_TN_SC_LINE : TN_SC_LINE;
	FB_TN_SC_ADD_SHADOW : TN_SC_ADD_SHADOW;
	FB_TN_SC_BOX : TN_SC_BOX;
	FB_TN_SC_WRITE_C : TN_SC_WRITE_C;
END_VAR
VAR
	in_ROW : INT;
	in_ROWS : INT;
	in_COL : INT;
	in_COLS : INT;
	in_index : INT;
	in_Count : INT;
	in_Scroll_Offset : INT;
	by_ATTR : BYTE;
END_VAR
VAR_IN_OUT
	Xus_TN_MENU_POPUP : us_TN_MENU_POPUP;
	Xus_TN_SCREEN : us_TN_SCREEN;
END_VAR

(*
version 1.1		06. apr 2011
programmer		ks
tested by			ks

TN_MENU_POPUP dient zur verwaltung und darstellung eines MENU-POPUP
*)

(* sicherstellen das rechteck immer innerhalb screen positioniert wird *)

IF (Xus_TN_MENU_POPUP.bo_Activ = FALSE) AND (Xus_TN_MENU_POPUP.bo_Create = TRUE) THEN
	Xus_TN_MENU_POPUP.bo_Activ := TRUE;
	Xus_TN_MENU_POPUP.bo_Create := FALSE;
	Xus_TN_MENU_POPUP.bo_Destroy := FALSE;
	Xus_TN_MENU_POPUP.bo_Update := TRUE;

  (* Sub-Menu-Texte *)

	Xus_TN_MENU_POPUP.in_Menu_E_Count := ELEMENT_COUNT(SEP:=BYTE#35,ELEMENT:=Xus_TN_MENU_POPUP.st_Menu_Text);

	(* Anzahl Zeilen (Sub-Menu-Texte) bestimmen *)
	Xus_TN_MENU_POPUP.in_Rows := Xus_TN_MENU_POPUP.in_Menu_E_Count;

	(* längsten Sub-Menu-Text suchen *)
	Xus_TN_MENU_POPUP.in_Cols := INT#00;

	FOR in_Count := INT#01 TO Xus_TN_MENU_POPUP.in_Rows DO;
		Xus_TN_MENU_POPUP.in_Cols:=MAX(LEN(ELEMENT_GET(SEP:=BYTE#35,POS:=in_Count - 1,ELEMENT:=Xus_TN_MENU_POPUP.st_Menu_Text)),Xus_TN_MENU_POPUP.in_Cols);
	END_FOR;

	(* Horizontale Position überprüfen und korrigieren *)
	IF (Xus_TN_MENU_POPUP.in_X + Xus_TN_MENU_POPUP.in_Cols) > INT#75 THEN
		Xus_TN_MENU_POPUP.in_X := INT#79 - Xus_TN_MENU_POPUP.in_Cols - INT#04;
	END_IF;

  (* Vertikale Position überprüfen und korrigieren *)
	IF (Xus_TN_MENU_POPUP.in_Y + Xus_TN_MENU_POPUP.in_ROWS) > INT#21 THEN
		Xus_TN_MENU_POPUP.in_Y := INT#23 - Xus_TN_MENU_POPUP.in_ROWS - INT#2;
	END_IF;

	Xus_TN_SCREEN.bo_Modal_Dialog := TRUE;

	(* Hintergrund sichern *)
	FB_TN_SC_AREA_SAVE(	Iin_X1 := Xus_TN_MENU_POPUP.in_X,
									Iin_Y1 := Xus_TN_MENU_POPUP.in_Y,
									Iin_X2 := Xus_TN_MENU_POPUP.in_X + Xus_TN_MENU_POPUP.in_Cols + INT#04,
									Iin_Y2 := Xus_TN_MENU_POPUP.in_Y + Xus_TN_MENU_POPUP.in_Rows + INT#02,
									Xus_TN_SCREEN := Xus_TN_SCREEN);

	(* Rahmen für Submenu zeichnen *)
	FB_TN_SC_BOX(	Iin_X1 := Xus_TN_MENU_POPUP.in_X,
					Iin_Y1 := Xus_TN_MENU_POPUP.in_Y,
					Iin_X2 := Xus_TN_MENU_POPUP.in_X + Xus_TN_MENU_POPUP.in_Cols + INT#03,
					Iin_Y2 := Xus_TN_MENU_POPUP.in_Y + Xus_TN_MENU_POPUP.in_Rows + INT#01,
					Iby_FILL := BYTE#32, (* Füllung *)
					Iin_BORDER := INT#01, (* Single-Line Border *)
					Iby_ATTR := Xus_TN_MENU_POPUP.by_Attr_oF,
					Xus_TN_SCREEN := Xus_TN_SCREEN);

	(* Shadow für Submenu zeichnen *)
	FB_TN_SC_ADD_SHADOW(Iin_X1 := Xus_TN_MENU_POPUP.in_X + INT#1,
						Iin_Y1 := Xus_TN_MENU_POPUP.in_Y + INT#1,
						Iin_X2 := Xus_TN_MENU_POPUP.in_X + Xus_TN_MENU_POPUP.in_Cols + INT#04,
						Iin_Y2 := Xus_TN_MENU_POPUP.in_Y + Xus_TN_MENU_POPUP.in_Rows + INT#02,
						Iin_OPTION := INT#00,
						Xus_TN_SCREEN := Xus_TN_SCREEN);

	(* Parameter laden *)
	in_COL := Xus_TN_MENU_POPUP.in_X;
	in_ROW := Xus_TN_MENU_POPUP.in_Y;
	in_ROWS := Xus_TN_MENU_POPUP.in_Rows;
	in_COLS := Xus_TN_MENU_POPUP.in_Cols;

	(* Trennlinien zeichnen *)
	in_COLS := in_COLS + INT#02; (* Text um 2 Zeichen verlängern *)

	FOR in_Count := INT#01 TO Xus_TN_MENU_POPUP.in_Menu_E_Count DO;
		in_ROW := in_ROW + INT#01;

		IF ELEMENT_GET(SEP:=BYTE#35,POS:=in_Count - 1,ELEMENT:=Xus_TN_MENU_POPUP.st_Menu_Text) = '-' THEN

			FB_TN_SC_LINE(	Iin_Y1 := in_ROW,
							Iin_X1 := in_COL,
							Iin_Y2 := in_ROW,
							Iin_X2 := in_COL + in_COLS + INT#01,
							Iby_ATTR := Xus_TN_MENU_POPUP.by_Attr_oF,
							Iby_BORDER := BYTE#01,
							Xus_TN_SCREEN := Xus_TN_SCREEN);
		END_IF;
	END_FOR;
END_IF;

IF (Xus_TN_MENU_POPUP.bo_Activ = TRUE) THEN

	CASE BYTE_TO_INT(Xus_TN_MENU_POPUP.by_Input_Exten_Code) OF

	65: (* Cursor oben *)
		in_Scroll_Offset := -1;
		Xus_TN_MENU_POPUP.bo_Update := TRUE;

	66: (* Cursor unten *)
		in_Scroll_Offset := 1;
		Xus_TN_MENU_POPUP.bo_Update := TRUE;

	13:  (* Enter *)
		Xus_TN_MENU_POPUP.bo_Destroy := TRUE;

	27:  (* Escape*)
		Xus_TN_MENU_POPUP.bo_Destroy := TRUE;
		Xus_TN_MENU_POPUP.in_Cur_Item := INT#00;

	67..68: (* Cursor links oder rechts *)
		Xus_TN_MENU_POPUP.bo_Destroy := TRUE;
		Xus_TN_MENU_POPUP.in_Cur_Item := INT#00;

	END_CASE;
END_IF;

(* POPUP-Menu updaten *)
IF (Xus_TN_MENU_POPUP.bo_Activ = TRUE) AND (Xus_TN_MENU_POPUP.bo_Update = TRUE) THEN

	Xus_TN_MENU_POPUP.bo_Update := FALSE;

	(* überprüfung + nächstes anwählbares Sub-Menu suchen *)
	in_index := Xus_TN_MENU_POPUP.in_Cur_Item;

	IF (in_index < INT#01) OR (in_index > Xus_TN_MENU_POPUP.in_Menu_E_Count) THEN
		in_Scroll_Offset := INT#01;
		in_index := Xus_TN_MENU_POPUP.in_Menu_E_Count;
	END_IF;

	(* aktueller Index steht auf Trennzeichen -> ändern *)
	IF ELEMENT_GET(SEP:=BYTE#35,POS:=in_index-1,ELEMENT:=Xus_TN_MENU_POPUP.st_Menu_Text) = '-' THEN
		in_Scroll_Offset := INT#01;
	END_IF;

	(* Scroll-Offset *)
	IF in_Scroll_Offset <> INT#00 THEN

		FOR in_Count := INT#01 TO Xus_TN_MENU_POPUP.in_Menu_E_Count DO;

			in_index:=OSCAT_BASIC.INC2(in_index,in_Scroll_Offset,1,Xus_TN_MENU_POPUP.in_Menu_E_Count);

			IF ELEMENT_GET(SEP:=BYTE#35,POS:=in_index - 1,ELEMENT:=Xus_TN_MENU_POPUP.st_Menu_Text) <> '-' THEN
				EXIT;
			END_IF;

		END_FOR;
	END_IF;

	Xus_TN_MENU_POPUP.in_Cur_Item := in_index;
	in_Scroll_Offset := INT#00;

	(* Parameter laden *)
	in_COL  := Xus_TN_MENU_POPUP.in_X;
	in_ROW  := Xus_TN_MENU_POPUP.in_Y;
	in_ROWS := Xus_TN_MENU_POPUP.in_Rows;
	in_COLS := Xus_TN_MENU_POPUP.in_Cols;

	(* SUB-MENU-Titel ausgeben *)
	in_COLS := in_COLS + INT#02; (* Text um 2 Zeichen verlängern *)

	FOR in_Count := INT#01 TO Xus_TN_MENU_POPUP.in_Menu_E_Count DO;

		in_ROW := in_ROW + INT#01;

		(* Zeichenfarbe bestimmen *)
		IF in_Count = Xus_TN_MENU_POPUP.in_Cur_Item THEN
			by_ATTR := Xus_TN_MENU_POPUP.by_Attr_mF;
		ELSE
			by_ATTR := Xus_TN_MENU_POPUP.by_Attr_oF;
		END_IF;

		FB_TN_SC_WRITE_C.Ist_STRING := ELEMENT_GET(SEP:=BYTE#35,POS:=in_Count - 1,ELEMENT:=Xus_TN_MENU_POPUP.st_Menu_Text);

		IF FB_TN_SC_WRITE_C.Ist_STRING <> '-' THEN

			FB_TN_SC_WRITE_C(	Iin_Y := in_ROW,
								Iin_X := in_COL + INT#01,
								Iby_ATTR := by_ATTR,
								Iin_LENGTH := in_COLS,
								Iin_OPTION := INT#02, (* Center *)
								Xus_TN_SCREEN := Xus_TN_SCREEN);
		END_IF;
	END_FOR;
END_IF;

(* POPUP-Menu entfernen (Destroy) *)
IF (Xus_TN_MENU_POPUP.bo_Activ = TRUE) AND (Xus_TN_MENU_POPUP.bo_Destroy = TRUE) THEN

	Xus_TN_MENU_POPUP.bo_Destroy := FALSE;
	Xus_TN_MENU_POPUP.bo_Activ := FALSE;

	(* alten Hintergrund aus Speicher wiederherstellen *)
	FB_TN_SC_AREA_RESTORE(Xus_TN_SCREEN := Xus_TN_SCREEN);

	Xus_TN_SCREEN.bo_Modal_Dialog := FALSE;
END_IF;

(* revision history

ks	06. apr. 2011	rev 1.1
	list_len und list_get durch element_count und element_get ersetzt

ks	10. mai. 2010	rev 1.0
	original version
*)

END_FUNCTION_BLOCK

// POUs/TELNET_VISION/TN_SC_AREA_SAVE
FUNCTION_BLOCK TN_SC_AREA_SAVE
VAR
	in_Offset_1 : INT;
	in_Offset_2 : INT;
	in_Y : INT;
	in_X : INT;
END_VAR
VAR_INPUT
	Iin_Y1 : INT;
	Iin_X1 : INT;
	Iin_Y2 : INT;
	Iin_X2 : INT;
END_VAR
VAR_IN_OUT
	Xus_TN_SCREEN : us_TN_SCREEN;
END_VAR

(*
version 1.0		10. mai 2010
programmer		ks
tested by		ks

TN_SC_AREA_SAVE sichert den angegebenen Bildschirmbereich in einem Buffer
*)

IF TN_SC_XY2_ERROR(Iin_X1,Iin_Y1,Iin_X2,Iin_Y2) THEN RETURN; END_IF;

(* Parameter ablegen *)
Xus_TN_SCREEN.bya_BACKUP[0] := BYTE#1;
Xus_TN_SCREEN.bya_BACKUP[1] := INT_TO_BYTE(Iin_X1);
Xus_TN_SCREEN.bya_BACKUP[2] := INT_TO_BYTE(Iin_Y1); 
Xus_TN_SCREEN.bya_BACKUP[3] := INT_TO_BYTE(Iin_X2);
Xus_TN_SCREEN.bya_BACKUP[4] := INT_TO_BYTE(Iin_Y2);

in_Offset_2 := 5;
(* CHAR und COLOR in BUFFER sichern *)
FOR in_Y := Iin_Y1 TO Iin_Y2 DO

	in_Offset_1 := (in_Y * 80) + Iin_X1;
	FOR in_X := Iin_X1 TO Iin_X2 DO
		Xus_TN_SCREEN.bya_BACKUP[in_Offset_2] := Xus_TN_SCREEN.bya_CHAR[in_Offset_1];
		in_Offset_2 := in_Offset_2 + INT#01;
		Xus_TN_SCREEN.bya_BACKUP[in_Offset_2] := Xus_TN_SCREEN.bya_COLOR[in_Offset_1];
		in_Offset_2 := in_Offset_2 + INT#01;
		in_Offset_1 := in_Offset_1 + INT#01;
	END_FOR;
END_FOR;

(* revision history
ks	10. mai. 2010	rev 1.0
	original version
*)

END_FUNCTION_BLOCK

// POUs/TELNET_VISION/TN_SC_XY2_ERROR
FUNCTION TN_SC_XY2_ERROR : BOOL
VAR_INPUT
	X1 : INT;
	Y1 : INT;
	X2 : INT;
	Y2 : INT;
END_VAR

(*
version 1.0		10. mai 2010
programmer		ks
tested by		ks

TN_SC_XY2_ERROR prüft ob die angegenene Koordinaten die einen rechteckigen Bereich angeben gültig sind 
*)

(* min und max werte prüfen *)
TN_SC_XY2_ERROR := Y1 < 0 OR X1 < 0 OR Y2 < 0 OR X2 < 0 OR Y1 > 23 OR X1 > 79 OR Y2 > 23 OR X2 > 79;

(* revision history
ks	10. mai. 2010	rev 1.0
	original version
*)

END_FUNCTION

// POUs/TELNET_VISION/TN_SC_AREA_RESTORE
FUNCTION_BLOCK TN_SC_AREA_RESTORE
VAR
	in_Offset_1 : INT;
	in_Offset_2 : INT;
	in_Y : INT;
	in_X : INT;
	in_Y1 : INT;
	in_X1 : INT;
	in_Y2 : INT;
	in_X2 : INT;
END_VAR
VAR_IN_OUT
	Xus_TN_SCREEN : us_TN_SCREEN;
END_VAR

(*
version 1.0		10. mai 2010
programmer		ks
tested by		ks

TN_SC_AREA_RESTORE stellt den zuvor gesicherten Bildschirmbereich wieder her
*)

IF Xus_TN_SCREEN.bya_BACKUP[0] > BYTE#00 THEN

	(* Parameter auslesen *)
	in_X1 := BYTE_TO_INT(Xus_TN_SCREEN.bya_BACKUP[1]);
	in_Y1 := BYTE_TO_INT(Xus_TN_SCREEN.bya_BACKUP[2]);
	in_X2 := BYTE_TO_INT(Xus_TN_SCREEN.bya_BACKUP[3]);
	in_Y2 := BYTE_TO_INT(Xus_TN_SCREEN.bya_BACKUP[4]);

	IF TN_SC_XY2_ERROR(in_X1,in_Y1,in_X2,in_Y2) THEN RETURN; END_IF;
	in_Offset_2 := 5;

	(* CHAR und COLOR von BUFFER wiederherstellen *)
	FOR in_Y := in_Y1 TO in_Y2 DO

		Xus_TN_SCREEN.bya_Line_Update[in_Y] := TRUE; (* Zeile zum Updaten freigeben *)
		in_Offset_1 := (in_Y * 80) + in_X1;

		FOR in_X := in_X1 TO in_X2 DO

			Xus_TN_SCREEN.bya_CHAR[in_Offset_1] := Xus_TN_SCREEN.bya_BACKUP[in_Offset_2];
			in_Offset_2 := in_Offset_2 + INT#01;

			Xus_TN_SCREEN.bya_COLOR[in_Offset_1] := Xus_TN_SCREEN.bya_BACKUP[in_Offset_2];
			in_Offset_2 := in_Offset_2 + INT#01;
			in_Offset_1 := in_Offset_1 + INT#01;

		END_FOR;
	END_FOR;

	(* Daten als ungültig markieren *)
	Xus_TN_SCREEN.bya_BACKUP[0] := BYTE#00;
END_IF;

(* revision history
ks	10. mai. 2010	rev 1.0
	original version
*)

END_FUNCTION_BLOCK

// POUs/TELNET_VISION/TN_SC_LINE
FUNCTION_BLOCK TN_SC_LINE
VAR
	by_Connect_Left_Char : BYTE;
	by_Connect_Right_Char : BYTE;
	by_Connect_Top_Char : BYTE;
	by_Connect_Bottom_Char : BYTE;
	by_Connect_Cruz_Char : BYTE;
	by_Vertikal_Line_Char : BYTE;
	by_Horzontal_Line_Char : BYTE;
	by_old_Char : BYTE;
	in_Offset_1 : INT;
	in_ROW_Index : INT;
	in_COL_Index : INT;
	by_Char : BYTE;
END_VAR
VAR_INPUT
	Iin_X1 : INT;
	Iin_Y1 : INT;
	Iin_X2 : INT;
	Iin_Y2 : INT;
	Iby_ATTR : BYTE;
	Iby_BORDER : BYTE;
END_VAR
VAR_IN_OUT
	Xus_TN_SCREEN : us_TN_SCREEN;
END_VAR

(*
version 1.0		10. mai 2010
programmer		ks
tested by		ks

TN_SC_LINE zeichnet horizontale und vertikale Linien
*)

IF TN_SC_XY2_ERROR(Iin_X1,Iin_Y1,Iin_X2,Iin_Y2) THEN RETURN; END_IF;

(* Bordertype bestimmen *)
IF Iby_Border = BYTE#01 THEN (* Single Line *)
	by_Connect_Top_Char := BYTE#16#C2;
	by_Connect_Bottom_Char := BYTE#16#C1;
	by_Connect_Left_Char := BYTE#16#C3;
	by_Connect_Right_Char := BYTE#16#B4;
	by_Horzontal_Line_Char := BYTE#16#C4;
	by_Vertikal_Line_Char := BYTE#16#B3;
	by_Connect_Cruz_Char := BYTE#16#C5;
ELSIF Iby_Border = BYTE#02 THEN	(* Double Linie *)
	by_Connect_Top_Char := BYTE#16#CB;
	by_Connect_Bottom_Char := BYTE#16#CA;
	by_Connect_Left_Char := BYTE#16#CC;
	by_Connect_Right_Char := BYTE#16#B9;
	by_Horzontal_Line_Char := BYTE#16#CD;
	by_Vertikal_Line_Char := BYTE#16#BA;
	by_Connect_Cruz_Char := BYTE#16#CE;
ELSE (* Full Linie *)
	by_Connect_Top_Char := Iby_Border;
	by_Connect_Bottom_Char := Iby_Border;
	by_Connect_Left_Char := Iby_Border;
	by_Connect_Right_Char := Iby_Border;
	by_Horzontal_Line_Char := Iby_Border;
	by_Vertikal_Line_Char := Iby_Border;
	by_Connect_Cruz_Char := Iby_Border;
END_IF;

(* Vertikale Linie zeichnen *)
IF Iin_X1 = Iin_X2 THEN
	in_Offset_1 := (Iin_Y1 * 80) + Iin_X1;
	FOR in_ROW_Index := Iin_Y1 TO Iin_Y2 DO
		by_old_Char := Xus_TN_SCREEN.bya_CHAR[in_Offset_1]; (* bestehendes Zeichen auslesen *)
		by_Char := by_Vertikal_Line_Char; (* Standardzeichen vorbelegen *)
		IF by_old_Char = by_Horzontal_Line_Char THEN (* Schnittpunkt erkannt *)
			IF in_ROW_Index = Iin_Y1 THEN (* Anfang der Linie behandeln *)
				by_Char := by_Connect_Top_Char;
			ELSIF in_ROW_Index = Iin_Y2 THEN (* Ende der Linie behandeln *)
				by_Char := by_Connect_Bottom_Char;
			ELSE (* Kreuzungspunkt behandeln *)
				by_Char := by_Connect_Cruz_Char;
			END_IF;
		END_IF;
		Xus_TN_SCREEN.bya_Line_Update[in_ROW_Index] := TRUE; (* Zeile zum Updaten freigeben *)
		Xus_TN_SCREEN.bya_CHAR[in_Offset_1] := by_Char;
		Xus_TN_SCREEN.bya_COLOR[in_Offset_1] := Iby_Attr;
		in_Offset_1 := in_Offset_1 + 80;
	END_FOR;

ELSIF Iin_Y1 = Iin_Y2 THEN (* Horzontale Linie zeichnen *)
	Xus_TN_SCREEN.bya_Line_Update[Iin_Y1] := TRUE; (* Zeile zum Updaten freigeben *)
	in_Offset_1 := (Iin_Y1 * 80) + Iin_X1;
	FOR in_COL_Index := Iin_X1 TO Iin_X2 DO
		by_old_Char := Xus_TN_SCREEN.bya_CHAR[in_Offset_1]; (* bestehendes Zeichen auslesen *)
		by_Char := by_Horzontal_Line_Char; (* Standardzeichen vorbelegen *)
		IF by_old_Char = by_Vertikal_Line_Char THEN (* Schnittpunkt erkannt *)
			IF in_COL_Index = Iin_X1 THEN (* Anfang der Linie behandeln *)
				by_Char := by_Connect_Left_Char;
			ELSIF in_COL_Index = Iin_X2 THEN (* Ende der Linie behandeln *)
				by_Char := by_Connect_Right_Char;
			ELSE (* Kreuzungspunkt behandeln *)
				by_Char := by_Connect_Cruz_Char;
			END_IF;
		END_IF;
		Xus_TN_SCREEN.bya_CHAR[in_Offset_1] := by_Char;
		Xus_TN_SCREEN.bya_COLOR[in_Offset_1] := Iby_Attr;
		in_Offset_1 := in_Offset_1 + 1;
	END_FOR;
END_IF;

(* revision history
ks	10. mai. 2010	rev 1.0
	original version
*)

END_FUNCTION_BLOCK

// POUs/TELNET_VISION/TN_SC_ADD_SHADOW
FUNCTION_BLOCK TN_SC_ADD_SHADOW
VAR
	in_Offset : INT;
	in_X : INT;
	in_Y : INT;
END_VAR
VAR_INPUT
	Iin_Y1 : INT;
	Iin_X1 : INT;
	Iin_Y2 : INT;
	Iin_X2 : INT;
	Iin_OPTION : INT;
END_VAR
VAR_IN_OUT
	Xus_TN_SCREEN : us_TN_SCREEN;
END_VAR

(*
version 1.0		10. mai 2010
programmer		ks
tested by		ks

TN_SC_ADD_SHADOW zeichnet auf der linken und unteren Seite eines rechteckigen Bereiches einen Schatten
*)

IF TN_SC_XY2_ERROR(Iin_X1,Iin_Y1,Iin_X2,Iin_Y2) THEN RETURN; END_IF;

IF Iin_Y1 < 0 OR Iin_X1 < 0 OR Iin_Y2 < 0 OR Iin_X2 < 0 THEN RETURN; END_IF; (* min werte prüfen *)
IF Iin_Y1 > 23 OR Iin_X1 > 79 OR Iin_Y2 > 23 OR Iin_X2 > 79 THEN RETURN; END_IF; (* max werte prüfen *)

in_Offset := (Iin_Y1 * 80) + Iin_X2;

IF Iin_OPTION = INT#00 THEN
	(* Schatten durch Farbanpassung erzeugen *)
	FOR in_Y := Iin_Y1 TO Iin_Y2 DO
		Xus_TN_SCREEN.bya_COLOR[in_Offset] := TN_SC_SHADOW_ATTR(Xus_TN_SCREEN.bya_COLOR[in_Offset]);
		in_Offset := in_Offset + 80;
		Xus_TN_SCREEN.bya_Line_Update[in_Y] := TRUE; (* Zeile für Update eintragen *)
	END_FOR;
ELSE
	(* Schatten durch Farbe Schwarz und Leerzeichen erzeugen *)
	FOR in_Y := Iin_Y1 TO Iin_Y2 DO
		Xus_TN_SCREEN.bya_COLOR[in_Offset] := BYTE#00;
		Xus_TN_SCREEN.bya_CHAR[in_Offset] := BYTE#32;
		in_Offset := in_Offset + 80;
		Xus_TN_SCREEN.bya_Line_Update[in_Y] := TRUE; (* Zeile für Update eintragen *)
	END_FOR;
END_IF;

in_Offset := (Iin_Y2 * 80) + Iin_X1;

IF Iin_OPTION = INT#00 THEN
	(* Schatten durch Farbanpassung erzeugen *)
	FOR in_X  := Iin_X1 TO Iin_X2 DO
		Xus_TN_SCREEN.bya_COLOR[in_Offset] := TN_SC_SHADOW_ATTR(Xus_TN_SCREEN.bya_COLOR[in_Offset]);
		in_Offset := in_Offset + 1;
	END_FOR;
ELSE
	(* Schatten durch Farbe Schwarz und Leerzeichen erzeugen *)
	FOR in_X  := Iin_X1 TO Iin_X2 DO
		Xus_TN_SCREEN.bya_COLOR[in_Offset] := BYTE#00;
		Xus_TN_SCREEN.bya_CHAR[in_Offset] := BYTE#32;
		in_Offset := in_Offset + 1;
	END_FOR;
END_IF;

(* revision history
ks	10. mai. 2010	rev 1.0
	original version
*)

END_FUNCTION_BLOCK

// POUs/TELNET_VISION/TN_SC_SHADOW_ATTR
FUNCTION TN_SC_SHADOW_ATTR : BYTE
VAR_INPUT
	Iby_ATTR : BYTE;
END_VAR

(*
version 1.0		10. mai 2010
programmer		ks
tested by		ks

TN_SC_SHADOW_ATTR berechnet aus einem normalen einem abgedunkelten Farbcode
*)

(* Background Farbe auf Schwarz ändern      *)
(* und dunkle Fordergrundfarben einschalten *)  
TN_SC_SHADOW_ATTR := ((Iby_ATTR AND BYTE#2#11110000) OR BYTE#2#00001000);

(* revision history
ks	10. mai. 2010	rev 1.0
	original version
*)

END_FUNCTION

// POUs/TELNET_VISION/TN_SC_BOX
FUNCTION_BLOCK TN_SC_BOX
VAR
	FB_TN_SC_FILL : TN_SC_FILL;
	by_BorderChar_L_T : BYTE;
	by_BorderChar_T : BYTE;
	by_BorderChar_B : BYTE;
	by_BorderChar_R_T : BYTE;
	by_BorderChar_L : BYTE;
	by_BorderChar_R : BYTE;
	by_BorderChar_L_B : BYTE;
	by_BorderChar_R_B : BYTE;
	in_Y : INT;
	in_X : INT;
	in_Border_Offset : INT;
	in_Offset_1 : INT;
	in_Offset_2 : INT;
END_VAR
VAR_INPUT
	Iin_Y1 : INT;
	Iin_X1 : INT;
	Iin_Y2 : INT;
	Iin_X2 : INT;
	Iby_FILL : BYTE;
	Iby_ATTR : BYTE;
	Iin_BORDER : INT;
END_VAR
VAR_IN_OUT
	Xus_TN_SCREEN : us_TN_SCREEN;
END_VAR

(*
version 1.0		10. mai 2010
programmer		ks
tested by		ks

TN_SC_BOX füllt einen rechteckigen Bereich mit einem Zeichen und zeichnet eine Umrandung
*)

IF TN_SC_XY2_ERROR(Iin_X1,Iin_Y1,Iin_X2,Iin_Y2) THEN RETURN; END_IF;

(* Bordertype bestimmen *)
CASE Iin_Border OF
0:
	in_Border_Offset := 0;
1:
	by_BorderChar_L_T := BYTE#218; (* links oben *)
	by_BorderChar_T := BYTE#196; (* oben *)
	by_BorderChar_R_T := BYTE#191; (* rechts oben *)
	by_BorderChar_L := BYTE#179; (* links *)
	by_BorderChar_R := BYTE#179; (* rechts *)
	by_BorderChar_B := BYTE#196; (* unten *)
	by_BorderChar_L_B := BYTE#217; (* links unten *)
	by_BorderChar_R_B := BYTE#192; (* rechts unten *)
	in_Border_Offset := 1;
 2:
	by_BorderChar_L_T := BYTE#201;
	by_BorderChar_T := BYTE#205;
	by_BorderChar_R_T := BYTE#187;
	by_BorderChar_L := BYTE#186;
	by_BorderChar_R := BYTE#186;
	by_BorderChar_B := BYTE#205;
	by_BorderChar_L_B := BYTE#188;
	by_BorderChar_R_B := BYTE#200;
	in_Border_Offset := 1;
ELSE
	by_BorderChar_L_T := BYTE#32;
	by_BorderChar_T := BYTE#32;
	by_BorderChar_R_T := BYTE#32;
	by_BorderChar_L := BYTE#32;
	by_BorderChar_R := BYTE#32;
	by_BorderChar_B := BYTE#32;
	by_BorderChar_L_B := BYTE#32;
	by_BorderChar_R_B := BYTE#32;
	in_Border_Offset := 1;

END_CASE;

IF Iby_FILL > BYTE#0 THEN (* FILL Zeichen vorhanden ? -> Box zeichnen *)

	(* Fill-Function um eine Zeichenreihe kleiner zeichnen *)
	FB_TN_SC_FILL(	Iin_Y1 := Iin_Y1 + in_Border_Offset,
					Iin_X1 := Iin_X1 + in_Border_Offset,
					Iin_Y2 := Iin_Y2 - in_Border_Offset,
					Iin_X2 := Iin_X2 - in_Border_Offset,
					Iby_CHAR := Iby_FILL,
					Iby_Attr := Iby_ATTR,
					Xus_TN_SCREEN := Xus_TN_SCREEN);
END_IF;

IF Iin_BORDER = 0 THEN RETURN; END_IF;

(* linken und rechten Rand ausgeben *)

in_Offset_1 := (Iin_Y1 * 80) + Iin_X1;
in_Offset_2 := (Iin_Y1 * 80) + Iin_X2;

FOR in_Y := Iin_Y1 TO Iin_Y2 DO

	(* Zeile zum Updaten freigeben *)
	Xus_TN_SCREEN.bya_Line_Update[in_Y] := TRUE;

	Xus_TN_SCREEN.bya_CHAR[in_Offset_1] := by_BorderChar_L;
	Xus_TN_SCREEN.bya_COLOR[in_Offset_1] := Iby_Attr;

	Xus_TN_SCREEN.bya_CHAR[in_Offset_2] := by_BorderChar_R;
	Xus_TN_SCREEN.bya_COLOR[in_Offset_2] := Iby_Attr;

	in_Offset_1 := in_Offset_1 + 80;
	in_Offset_2 := in_Offset_2 + 80;

END_FOR;

(* unteren und oberen Rand ausgeben *)
in_Offset_1 := (Iin_Y1 * 80) + Iin_X1;
in_Offset_2 := (Iin_Y2 * 80) + Iin_X1;

FOR in_X := Iin_X1 TO Iin_X2 DO

	Xus_TN_SCREEN.bya_CHAR[in_Offset_1] := by_BorderChar_T;
	Xus_TN_SCREEN.bya_COLOR[in_Offset_1] := Iby_Attr;

	Xus_TN_SCREEN.bya_CHAR[in_Offset_2] := by_BorderChar_B;
	Xus_TN_SCREEN.bya_COLOR[in_Offset_2] := Iby_Attr;

	in_Offset_1 := in_Offset_1 + INT#1;
	in_Offset_2 := in_Offset_2 + INT#1;

END_FOR;

(* linke obere Ecke ausgeben *)
in_Offset_1 := (Iin_Y1 * 80) + Iin_X1;
Xus_TN_SCREEN.bya_CHAR[in_Offset_1] := by_BorderChar_L_T;
Xus_TN_SCREEN.bya_COLOR[in_Offset_1] := Iby_Attr;

(* rechte obere Ecke ausgeben *)
in_Offset_1 := (Iin_Y1 * 80) + Iin_X2;
Xus_TN_SCREEN.bya_CHAR[in_Offset_1] := by_BorderChar_R_T;
Xus_TN_SCREEN.bya_COLOR[in_Offset_1] := Iby_Attr;

(* linke untere Ecke ausgeben *)
in_Offset_1 := (Iin_Y2 * 80) + Iin_X1;
Xus_TN_SCREEN.bya_CHAR[in_Offset_1] := by_BorderChar_R_B;
Xus_TN_SCREEN.bya_COLOR[in_Offset_1] := Iby_Attr;

(* rechte untere Ecke ausgeben *)
in_Offset_1 := (Iin_Y2 * 80) + Iin_X2;
Xus_TN_SCREEN.bya_CHAR[in_Offset_1] := by_BorderChar_L_B;
Xus_TN_SCREEN.bya_COLOR[in_Offset_1] := Iby_Attr;

(* revision history
ks	10. mai. 2010	rev 1.0
	original version
*)

END_FUNCTION_BLOCK

// POUs/TELNET_VISION/TN_SC_FILL
FUNCTION_BLOCK TN_SC_FILL
VAR
	in_X : INT;
	in_Y : INT;
	in_Offset : INT;
END_VAR
VAR_INPUT
	Iin_Y1 : INT;
	Iin_X1 : INT;
	Iin_Y2 : INT;
	Iin_X2 : INT;
	Iby_CHAR : BYTE;
	Iby_Attr : BYTE;
END_VAR
VAR_IN_OUT
	Xus_TN_SCREEN : us_TN_SCREEN;
END_VAR

(*
version 1.0		10. mai 2010
programmer		ks
tested by		ks

TN_SC_FILL füllt einen rechteckigen Bereich mit einem Zeichen
*)

IF TN_SC_XY2_ERROR(Iin_X1,Iin_Y1,Iin_X2,Iin_Y2) THEN RETURN; END_IF;

FOR in_Y := Iin_Y1 TO Iin_Y2 DO
	Xus_TN_SCREEN.bya_Line_Update[in_Y] := TRUE; (* Zeile zum Updaten freigeben *)
	in_Offset := (in_Y * 80) + Iin_X1;
	FOR in_X := Iin_X1 TO Iin_X2 DO
		Xus_TN_SCREEN.bya_CHAR[in_Offset]  := Iby_CHAR; (* Zeichen eintragen *)
		Xus_TN_SCREEN.bya_COLOR[in_Offset] := Iby_Attr; (* Farbe eintragen *)
		in_Offset := in_Offset + 1;
	END_FOR;
END_FOR;

(* revision history
ks	10. mai. 2010	rev 1.0
	original version
*)

END_FUNCTION_BLOCK

// POUs/TELNET_VISION/TN_SC_WRITE_C
FUNCTION_BLOCK TN_SC_WRITE_C
VAR
	FB_TN_SC_WRITE : TN_SC_WRITE;
END_VAR
VAR_INPUT
	Iin_Y : INT;
	Iin_X : INT;
	Iby_ATTR : BYTE;
	Ist_STRING : STRING;
	Iin_LENGTH : INT;
	Iin_OPTION : INT;
END_VAR
VAR_IN_OUT
	Xus_TN_SCREEN : us_TN_SCREEN;
END_VAR

(*
version 1.0		10. mai 2010
programmer		ks
tested by		ks

TN_SC_WRITE_C korrigiert die Textlänge und schreibt den Text an die angegebenen Koordinate
*)

(* Text ausgeben *)
FB_TN_SC_WRITE( Iin_Y := Iin_Y,
				Iin_X := Iin_X,
				Iby_ATTR := Iby_ATTR,
				Ist_STRING := OSCAT_BASIC.FIX(str:=Ist_STRING,L:=Iin_LENGTH,C:=BYTE#32,M:=Iin_OPTION),
				Xus_TN_SCREEN := Xus_TN_SCREEN);

(* revision history
ks	10. mai. 2010	rev 1.0
	original version
*)

END_FUNCTION_BLOCK

// POUs/TELNET_VISION/TN_SC_WRITE
FUNCTION_BLOCK TN_SC_WRITE
VAR
	bo_Color : BOOL;
	in_Offset : INT;
	in_Char_Index : INT;
	in_String_Length : INT;
END_VAR
VAR_INPUT
	Iin_Y : INT;
	Iin_X : INT;
	Iby_ATTR : BYTE;
	Ist_STRING : STRING;
END_VAR
VAR_IN_OUT
	Xus_TN_SCREEN : us_TN_SCREEN;
END_VAR

(*
version 1.0		10. mai 2010
programmer		ks
tested by		ks

TN_SC_WRITE schreibt einem Text an die angegebene Koordinate
*)

in_String_Length := LEN(Ist_STRING);
IF TN_SC_XY_ERROR(Iin_X + in_String_Length - 1,Iin_Y) THEN RETURN; END_IF;
Xus_TN_SCREEN.bya_Line_Update[Iin_Y] := TRUE; (* Zeile zum Updaten freigeben *)
in_Offset := (Iin_Y * 80) + Iin_X; (* Offset des ersten Zeichen berechnen *)
bo_Color := Iby_ATTR <> BYTE#00;

(* Zeichen und Attribute des String kopieren *)
FOR in_Char_Index := 1 TO in_String_Length DO
	IF bo_Color THEN Xus_TN_SCREEN.bya_COLOR[in_Offset] := Iby_ATTR; END_IF;
	Xus_TN_SCREEN.bya_CHAR[in_Offset] := OSCAT_BASIC.CODE(STR:=Ist_STRING,POS:=in_Char_Index);
	in_Offset := in_Offset + INT#1;
END_FOR;

Xus_TN_SCREEN.in_EOS_Offset := in_Offset; (* End of String Offset sichern *)

(* revision history
ks	10. mai. 2010	rev 1.0
	original version
*)

END_FUNCTION_BLOCK

// POUs/TELNET_VISION/TN_SC_XY_ERROR
FUNCTION TN_SC_XY_ERROR : BOOL
VAR_INPUT
	X : INT;
	Y : INT;
END_VAR

(*
version 1.0		10. mai 2010
programmer		ks
tested by		ks

TN_SC_XY_ERROR prüft ob die angegenene Koordinaten gültig sind 
*)

(* min und max werte prüfen *)
TN_SC_XY_ERROR := Y < 0 OR X < 0 OR Y > 23 OR X > 79;

(* revision history
ks	10. mai. 2010	rev 1.0
	original version
*)

END_FUNCTION

// POUs/TELNET_VISION/TN_INPUT_SELECT_TEXT
FUNCTION_BLOCK TN_INPUT_SELECT_TEXT
VAR
	in_count : INT;
	by_Attr : BYTE;
	st_String : STRING;
END_VAR
VAR
	FB_TN_SC_WRITE : TN_SC_WRITE;
END_VAR
VAR_IN_OUT
	Xus_TN_SCREEN : us_TN_SCREEN;
	Xus_TN_INPUT_CONTROL_DATA : us_TN_INPUT_CONTROL_DATA;
END_VAR

(*
version 1.1		06. apr 2011
programmer		ks
tested by			ks

TN_SELECT_TEXT dient zur verwaltung und darstellung einer Elementeauswahl
*)

(* Benutzereingabe auswerten -> Selektion Text n *)
IF Xus_TN_INPUT_CONTROL_DATA.bo_Focus = TRUE THEN

(* Leertaste-Taste auswerten *)
	IF Xus_TN_INPUT_CONTROL_DATA.by_Input_ASCII_Code = BYTE#32 THEN
		Xus_TN_INPUT_CONTROL_DATA.in_selected := Xus_TN_INPUT_CONTROL_DATA.in_selected + INT#01; 
		Xus_TN_INPUT_CONTROL_DATA.bo_Update_Input := TRUE;
	END_IF;
 
	(* Return-Taste auswerten *)
	IF Xus_TN_INPUT_CONTROL_DATA.by_Input_Exten_Code = BYTE#13 THEN
		Xus_TN_INPUT_CONTROL_DATA.bo_Input_Entered := TRUE;
	END_IF;

END_IF;

(* Aktualisierung der Anzeige *)
IF (Xus_TN_INPUT_CONTROL_DATA.bo_Update_Input = TRUE) OR (Xus_TN_INPUT_CONTROL_DATA.bo_Update_All = TRUE) THEN

	(* Title-Text ausgeben *)
	IF Xus_TN_INPUT_CONTROL_DATA.bo_Update_All = TRUE THEN

		IF (Xus_TN_INPUT_CONTROL_DATA.in_Title_X_Offset = INT#00) AND (Xus_TN_INPUT_CONTROL_DATA.in_Title_Y_Offset = INT#00) THEN
			(* wenn Offset X,Y =0 dann Titlestring links vom Element positionieren *)
			FB_TN_SC_WRITE.Iin_Y := Xus_TN_INPUT_CONTROL_DATA.in_Y;
			FB_TN_SC_WRITE.Iin_X := Xus_TN_INPUT_CONTROL_DATA.in_X - LEN(Xus_TN_INPUT_CONTROL_DATA.st_Title_String);

		ELSE
			(* Title-Text durch Row, Color-Offset ausgeben *)
			FB_TN_SC_WRITE.Iin_Y := Xus_TN_INPUT_CONTROL_DATA.in_Y + Xus_TN_INPUT_CONTROL_DATA.in_Title_Y_Offset;
			FB_TN_SC_WRITE.Iin_X := Xus_TN_INPUT_CONTROL_DATA.in_X + Xus_TN_INPUT_CONTROL_DATA.in_Title_X_Offset;
		END_IF;

		(* Title-Text durch Row, Color-Offset ausgeben *)
		FB_TN_SC_WRITE(	Iby_ATTR := Xus_TN_INPUT_CONTROL_DATA.by_Title_Attr,
						Ist_STRING := Xus_TN_INPUT_CONTROL_DATA.st_Title_String,
						Xus_TN_SCREEN := Xus_TN_SCREEN);

	END_IF;

	(* Eingabezeile verarbeiten *)

	(* Anzahl der Elemente bestimmen *)
	in_count := ELEMENT_COUNT(SEP:=BYTE#35,ELEMENT:=Xus_TN_INPUT_CONTROL_DATA.st_Input_Data);

	IF in_Count > INT#00 THEN

		IF Xus_TN_INPUT_CONTROL_DATA.in_selected < INT#1 THEN
			Xus_TN_INPUT_CONTROL_DATA.in_selected := INT#01;
		END_IF;

		IF Xus_TN_INPUT_CONTROL_DATA.in_selected > in_count THEN
			Xus_TN_INPUT_CONTROL_DATA.in_selected := INT#01;
		END_IF;

		st_String := ELEMENT_GET(SEP:=BYTE#35,POS:=Xus_TN_INPUT_CONTROL_DATA.in_selected - 1,ELEMENT:=Xus_TN_INPUT_CONTROL_DATA.st_Input_Data);

		st_String := OSCAT_BASIC.FIX(	str:=st_String,
							L:=LEN(Xus_TN_INPUT_CONTROL_DATA.st_Input_Mask),
							C:=BYTE#32,
							M:=Xus_TN_INPUT_CONTROL_DATA.in_Input_Option);

		Xus_TN_INPUT_CONTROL_DATA.st_Input_String := st_String;

		IF Xus_TN_INPUT_CONTROL_DATA.bo_Focus = TRUE THEN
			by_Attr := Xus_TN_INPUT_CONTROL_DATA.by_Attr_mF;
		ELSE
			by_Attr := Xus_TN_INPUT_CONTROL_DATA.by_Attr_oF;
		END_IF;

		FB_TN_SC_WRITE(	Iin_Y := Xus_TN_INPUT_CONTROL_DATA.in_Y,
						Iin_X := Xus_TN_INPUT_CONTROL_DATA.in_X,
						Iby_ATTR := by_Attr,
						Ist_STRING := st_String,
						Xus_TN_SCREEN := Xus_TN_SCREEN);
	END_IF;

	(* Cursor auf aktuelle Position setzen *)
	Xus_TN_INPUT_CONTROL_DATA.in_Cursor_Y := Xus_TN_INPUT_CONTROL_DATA.in_Y;
	Xus_TN_INPUT_CONTROL_DATA.in_Cursor_X := Xus_TN_INPUT_CONTROL_DATA.in_X;

	(* Update-Flag's rücksetzen *)
	Xus_TN_INPUT_CONTROL_DATA.bo_Update_All := FALSE;
	Xus_TN_INPUT_CONTROL_DATA.bo_Update_Input := FALSE;

END_IF;

(* revision history

ks	06. apr. 2011	rev 1.1
	list_len und list_get durch element_count und element_get ersetzt

ks	10. mai. 2010	rev 1.0
	original version
*)

END_FUNCTION_BLOCK

// POUs/TELNET_VISION/TN_INPUT_EDIT_LINE
FUNCTION_BLOCK TN_INPUT_EDIT_LINE
VAR
	in_count : INT;
	in_Count_End : INT;
	in_CursorOffset : INT;
	by_Attr : BYTE;
	st_String : STRING;
	bo_Pos_Found : BOOL;
	st_CHAR : STRING(1);
	in_old_charpos : INT;
END_VAR
VAR
	FB_TN_SC_WRITE : TN_SC_WRITE;
END_VAR
VAR_IN_OUT
	Xus_TN_SCREEN : us_TN_SCREEN;
	Xus_TN_INPUT_CONTROL_DATA : us_TN_INPUT_CONTROL_DATA;
END_VAR

(*
version 1.0		10. mai 2010
programmer		ks
tested by		ks

TN_INPUT_EDIT_LINE ermöglicht die Eingabe von Texten durch eine Editierbare Eingabezeile
*)

(* Cursorsteuerung rücksetzen *)
in_CursorOffset := INT#0;

IF Xus_TN_INPUT_CONTROL_DATA.bo_Focus = TRUE THEN

	(* Texteingabe erkannt ? *)
	IF Xus_TN_INPUT_CONTROL_DATA.by_Input_ASCII_Code > BYTE#0 THEN

		IF (Xus_TN_INPUT_CONTROL_DATA.bo_Input_Only_Num = TRUE AND Xus_TN_INPUT_CONTROL_DATA.bo_Input_ASCII_IsNum = TRUE)
			OR (Xus_TN_INPUT_CONTROL_DATA.bo_Input_Only_Num = FALSE) THEN

			(* ASCII Wert in einen String wandeln *)
			st_CHAR := OSCAT_BASIC.CHR_TO_STRING(C:=Xus_TN_INPUT_CONTROL_DATA.by_Input_ASCII_Code);

			(* Eingabe übernehmen *)
			Xus_TN_INPUT_CONTROL_DATA.st_Input_Data := REPLACE(Xus_TN_INPUT_CONTROL_DATA.st_Input_Data,
			st_CHAR,INT#1,Xus_TN_INPUT_CONTROL_DATA.in_Cursor_Pos);

			in_CursorOffset := INT#1;
			Xus_TN_INPUT_CONTROL_DATA.bo_Update_Input := TRUE;
		END_IF;
	END_IF;

	CASE BYTE_TO_INT(Xus_TN_INPUT_CONTROL_DATA.by_Input_Exten_Code) OF

	67: (* Cursor rechts gedrückt *)
		in_CursorOffset := INT#1;

	68: (* Cursor links gedrückt *)
		in_CursorOffset := -1;

	08: (* Backspace gedrückt *)
		Xus_TN_INPUT_CONTROL_DATA.st_Input_Data := REPLACE(Xus_TN_INPUT_CONTROL_DATA.st_Input_Data, ' ', 1,Xus_TN_INPUT_CONTROL_DATA.in_Cursor_Pos);
		Xus_TN_INPUT_CONTROL_DATA.bo_Update_Input := TRUE;
		in_CursorOffset := -1;

	13: (* Enter-Taste gedrückt *)
		IF LEN(Xus_TN_INPUT_CONTROL_DATA.st_Input_Mask) > INT#00 THEN
			(* Eingabestring übernehmen *)
			Xus_TN_INPUT_CONTROL_DATA.st_Input_String := Xus_TN_INPUT_CONTROL_DATA.st_Input_Data;

			(* Eingabestring -> links und rechts Leerzeichen entfernen *)
			Xus_TN_INPUT_CONTROL_DATA.st_Input_String := OSCAT_BASIC.TRIME(str:=Xus_TN_INPUT_CONTROL_DATA.st_Input_String);
			Xus_TN_INPUT_CONTROL_DATA.bo_Input_Entered := TRUE;

			(* neue Eingabe vorbereiten *)
			Xus_TN_INPUT_CONTROL_DATA.st_Input_Data := Xus_TN_INPUT_CONTROL_DATA.st_Input_Mask;

			Xus_TN_INPUT_CONTROL_DATA.in_Cursor_Pos := INT#1;
			Xus_TN_INPUT_CONTROL_DATA.bo_Update_Input := TRUE;

			(* suche erstes Position in Eingabemaske *)
			st_CHAR := MID(Xus_TN_INPUT_CONTROL_DATA.st_Input_Mask,1,Xus_TN_INPUT_CONTROL_DATA.in_Cursor_Pos);
			IF st_CHAR <> ' ' THEN
				(* nächsten Eingabeposition suchen *)
				in_CursorOffset := INT#1;
			END_IF;
		END_IF;
	END_CASE;
END_IF;

(* Cursor richtung rechts bewegen                                   *)
IF (in_CursorOffset > INT#0) OR (Xus_TN_INPUT_CONTROL_DATA.in_Cursor_Pos = INT#0) THEN
	bo_Pos_Found := FALSE;

	in_Count := Xus_TN_INPUT_CONTROL_DATA.in_Cursor_Pos + INT#1;
	in_Count_End := LEN(Xus_TN_INPUT_CONTROL_DATA.st_Input_Mask);

	WHILE (in_count <= in_Count_End) AND (bo_Pos_Found = FALSE) DO

		st_CHAR := MID(Xus_TN_INPUT_CONTROL_DATA.st_Input_Mask,1,in_count);
		IF st_CHAR = ' ' THEN
			Xus_TN_INPUT_CONTROL_DATA.in_Cursor_Pos := in_count;
			Xus_TN_INPUT_CONTROL_DATA.bo_Update_Input := TRUE;
			bo_Pos_Found := TRUE;
		END_IF;

		in_count := in_count + INT#1;

	END_WHILE;
END_IF;

(* Cursor richtung links bewegen *)
IF in_CursorOffset < INT#0 THEN
	bo_Pos_Found := FALSE;

	in_Count     := Xus_TN_INPUT_CONTROL_DATA.in_Cursor_Pos - INT#01;
	in_Count_End := INT#1;

	WHILE (in_count >= in_Count_End) AND (bo_Pos_Found = FALSE) DO

		st_CHAR := MID(Xus_TN_INPUT_CONTROL_DATA.st_Input_Mask,1,in_count);
		IF st_CHAR = ' ' THEN
			Xus_TN_INPUT_CONTROL_DATA.in_Cursor_Pos := in_count;
			Xus_TN_INPUT_CONTROL_DATA.bo_Update_Input := TRUE;
			bo_Pos_Found := TRUE;
		END_IF;

		in_count := in_count - INT#1;
	END_WHILE;
END_IF;

(* maximale Cursorposition ? *)
IF Xus_TN_INPUT_CONTROL_DATA.in_Cursor_Pos > LEN(Xus_TN_INPUT_CONTROL_DATA.st_Input_Data) THEN
	Xus_TN_INPUT_CONTROL_DATA.in_Cursor_Pos := LEN(Xus_TN_INPUT_CONTROL_DATA.st_Input_Data);
	Xus_TN_INPUT_CONTROL_DATA.bo_Update_Input := TRUE;
END_IF;

(* minimale Cursorposition ? *)
IF Xus_TN_INPUT_CONTROL_DATA.in_Cursor_Pos < INT#1 THEN
	Xus_TN_INPUT_CONTROL_DATA.in_Cursor_Pos := INT#1;
	Xus_TN_INPUT_CONTROL_DATA.bo_Update_Input := TRUE;
END_IF;

(* Aktualisierung der Anzeige *)
IF (Xus_TN_INPUT_CONTROL_DATA.bo_Update_Input = TRUE) OR (Xus_TN_INPUT_CONTROL_DATA.bo_Update_All = TRUE) THEN

	(* Title-Text ausgeben *)
	IF (Xus_TN_INPUT_CONTROL_DATA.bo_Update_All = TRUE) THEN

		IF (Xus_TN_INPUT_CONTROL_DATA.in_Title_X_Offset = INT#00) AND (Xus_TN_INPUT_CONTROL_DATA.in_Title_Y_Offset = INT#00) THEN
			(* wenn Offset X,Y =0 dann Titlestring links vom Element positionieren *)
			FB_TN_SC_WRITE.Iin_Y := Xus_TN_INPUT_CONTROL_DATA.in_Y;
			FB_TN_SC_WRITE.Iin_X := Xus_TN_INPUT_CONTROL_DATA.in_X - LEN(Xus_TN_INPUT_CONTROL_DATA.st_Title_String);
		ELSE
			(* Title-Text durch Row, Color-Offset ausgeben *)
			FB_TN_SC_WRITE.Iin_Y := Xus_TN_INPUT_CONTROL_DATA.in_Y + Xus_TN_INPUT_CONTROL_DATA.in_Title_Y_Offset;
			FB_TN_SC_WRITE.Iin_X := Xus_TN_INPUT_CONTROL_DATA.in_X + Xus_TN_INPUT_CONTROL_DATA.in_Title_X_Offset;
		END_IF;

		(* Title-Text durch Row, Color-Offset ausgeben *)
		FB_TN_SC_WRITE(	Iby_ATTR := Xus_TN_INPUT_CONTROL_DATA.by_Title_Attr,
						Ist_STRING := Xus_TN_INPUT_CONTROL_DATA.st_Title_String,
						Xus_TN_SCREEN := Xus_TN_SCREEN);
	END_IF;

	(* Eingabetext ausgeben *)
	IF (Xus_TN_INPUT_CONTROL_DATA.bo_Input_Hidden = TRUE) THEN

		st_String := '';

		IF LEN(Xus_TN_INPUT_CONTROL_DATA.st_Input_Data) = LEN(Xus_TN_INPUT_CONTROL_DATA.st_Input_Mask) THEN
			(* Eingabemodus: HIDDEN *)
			FOR in_count := 1 TO LEN(Xus_TN_INPUT_CONTROL_DATA.st_Input_Data) DO

				(* Zeichen aus Eingabemaske lesen *)
				st_CHAR := MID(Xus_TN_INPUT_CONTROL_DATA.st_Input_Mask,1,in_count);

				(* Eingabe oder Maskenzeichen ausgeben *)
				IF st_CHAR = ' ' THEN

					(* Zeichen aus Eingabedata lesen *)
					st_CHAR := MID(Xus_TN_INPUT_CONTROL_DATA.st_Input_Data,1,in_count);

					IF st_CHAR = ' ' THEN
						(* Leerzeichen ausgeben *)
						st_String := CONCAT(st_String, ' ');

					ELSE
						(* verdecktes Zeichen ausgeben *)
						st_String := CONCAT(st_String, '*');

					END_IF;

				ELSE
					(* Zeichen aus Eingabemaske übernehmen *)
					st_CHAR := MID(Xus_TN_INPUT_CONTROL_DATA.st_Input_Data,1,in_count);
					st_String := CONCAT(st_String,st_CHAR);

				END_IF;
			END_FOR;
		END_IF;
	ELSE

		(* Eingabemodus: NORMAL *)
		st_String := Xus_TN_INPUT_CONTROL_DATA.st_Input_Data;

	END_IF;

	(* String ausgeben *)

	IF Xus_TN_INPUT_CONTROL_DATA.bo_Focus = TRUE THEN
		by_Attr := Xus_TN_INPUT_CONTROL_DATA.by_Attr_mF;
	ELSE
		by_Attr := Xus_TN_INPUT_CONTROL_DATA.by_Attr_oF;
	END_IF;

	FB_TN_SC_WRITE(	Iin_Y := Xus_TN_INPUT_CONTROL_DATA.in_Y,
					Iin_X := Xus_TN_INPUT_CONTROL_DATA.in_X,
					Iby_ATTR := by_Attr,
					Ist_STRING := st_String,
					Xus_TN_SCREEN := Xus_TN_SCREEN);

	(* Cursor auf aktuelle Position setzen *)
	Xus_TN_INPUT_CONTROL_DATA.in_Cursor_Y := Xus_TN_INPUT_CONTROL_DATA.in_Y;
	Xus_TN_INPUT_CONTROL_DATA.in_Cursor_X := Xus_TN_INPUT_CONTROL_DATA.in_X + Xus_TN_INPUT_CONTROL_DATA.in_Cursor_Pos - INT#1;

	in_old_charpos := INT#0;

	(* Update-Flag's rücksetzen *)
	Xus_TN_INPUT_CONTROL_DATA.bo_Update_All := FALSE;
	Xus_TN_INPUT_CONTROL_DATA.bo_Update_Input := FALSE;
END_IF;

(* revision history
ks	10. mai. 2010	rev 1.0
	original version
*)

END_FUNCTION_BLOCK

// POUs/TELNET_VISION/TN_INPUT_MENU_BAR
FUNCTION_BLOCK TN_INPUT_MENU_BAR
VAR
	FB_TN_INPUT_MENU_POPUP : TN_INPUT_MENU_POPUP;
	us_TN_MENU_POPUP : us_TN_MENU_POPUP;
	FB_TN_SC_WRITE_C : TN_SC_WRITE_C;
END_VAR
VAR
	in_ROW : INT;
	in_COL : INT;
	in_TITLE_Length : INT;
	st_MENU_BAR : STRING(OSCAT_BASIC.STRING_LENGTH);
	st_MENU_TITLE : STRING;
	in_Count : INT;
	in_Index : INT;
	by_New_KeyCode : BYTE;
	in_Scroll_Offset : INT;
	by_ATTR : BYTE;
	bo_Reset_Position :	BOOL;
END_VAR
VAR_IN_OUT
	Xus_TN_MENU : us_TN_MENU;
	Xus_TN_SCREEN : us_TN_SCREEN;
END_VAR

(*
version 1.1		06. apr 2011
programmer		ks
tested by			ks

TN_MENU_BAR ermöglicht die verwaltung und darstellung einer MENU-BAR
*)

(* sicherstellen das rechteck immer innerhalb screen positioniert wird *)

IF (Xus_TN_MENU.in_State = INT#00) AND (Xus_TN_MENU.bo_Create = TRUE) THEN
	Xus_TN_MENU.in_State := INT#01;
	Xus_TN_MENU.bo_Create := FALSE;
	Xus_TN_MENU.in_Menu_Selected := INT#00;
	Xus_TN_MENU.bo_Update := TRUE;
	bo_Reset_Position := TRUE;

	(* Menu-Bar - Hauptmenue *)
	st_MENU_BAR := ELEMENT_GET(SEP:=BYTE#37,POS:=0,ELEMENT:=Xus_TN_MENU.st_MENU_TEXT);

	(* Menu-Bar - Anzahl der Elemente bestimmen *)
	Xus_TN_MENU.in_Menu_E_Count := ELEMENT_COUNT(SEP:=BYTE#35,ELEMENT:=st_MENU_BAR);

END_IF;

(* Keycode ablegen *)
by_New_KeyCode := Xus_TN_SCREEN.by_Input_Exten_Code;

(* Popup-Menu Tastensteuerung (nur Cursor oben + unten zulassen *)
IF (by_New_KeyCode = BYTE#65) OR (by_New_KeyCode = BYTE#66) THEN
	us_TN_MENU_POPUP.by_Input_Exten_Code := by_New_KeyCode;
ELSE
	us_TN_MENU_POPUP.by_Input_Exten_Code := BYTE#00;
END_IF;

(* Escape *)
IF (by_New_KeyCode = BYTE#27) THEN
	(* Menu war inaktiv -> Escape -> Menu aktivieren *)
	IF (Xus_TN_MENU.in_State = INT#01) AND (Xus_TN_SCREEN.bo_Modal_Dialog = FALSE) THEN
		Xus_TN_MENU.in_State := INT#02;
		Xus_TN_MENU.bo_Update := TRUE;
		Xus_TN_MENU.in_Menu_Selected := INT#00;

		Xus_TN_SCREEN.bo_Menue_Bar_Dialog := TRUE;

		(* Menu war aktiv -> Escape -> Menu deaktivieren *)
	ELSIF (Xus_TN_MENU.in_State = INT#02) THEN
		us_TN_MENU_POPUP.bo_Destroy := TRUE;
		Xus_TN_MENU.bo_Update := TRUE;
		Xus_TN_MENU.in_State := INT#01;
		bo_Reset_Position := TRUE;

		Xus_TN_SCREEN.bo_Menue_Bar_Dialog := FALSE;
	END_IF;
END_IF;

(* Menu aktiv *)
IF (Xus_TN_MENU.in_State = INT#02) THEN

	(* Return *)
	IF (by_New_KeyCode = BYTE#13)  THEN
		us_TN_MENU_POPUP.bo_Destroy := TRUE;
		Xus_TN_MENU.bo_Update := TRUE;
		Xus_TN_MENU.in_State := INT#01;
		bo_Reset_Position := TRUE;
		Xus_TN_MENU.in_Menu_Selected := (Xus_TN_MENU.in_Cur_Menu_Item * INT#10) + Xus_TN_MENU.in_Cur_Sub_Item;
		Xus_TN_SCREEN.by_Input_Exten_Code := BYTE#00;

		Xus_TN_SCREEN.bo_Menue_Bar_Dialog := FALSE;

		(* Destroy-Befehl -> Popup-Menu beenden *)
	ELSIF (Xus_TN_MENU.bo_Destroy = TRUE) THEN
		us_TN_MENU_POPUP.bo_Destroy := TRUE;
		Xus_TN_MENU.bo_Update := TRUE;
		Xus_TN_MENU.in_State := INT#01;
		bo_Reset_Position := TRUE;
		Xus_TN_MENU.in_Menu_Selected := INT#00;
		Xus_TN_SCREEN.by_Input_Exten_Code := BYTE#00;

		Xus_TN_SCREEN.bo_Menue_Bar_Dialog := FALSE;

	END_IF;

	IF (by_New_KeyCode = BYTE#67) THEN (* Cursor rechts *)
		in_Scroll_Offset := INT#1;
		Xus_TN_MENU.bo_Update := TRUE;
		Xus_TN_SCREEN.by_Input_Exten_Code := BYTE#00;

	ELSIF (by_New_KeyCode = BYTE#68) THEN (* Cursor links *)
		in_Scroll_Offset := -1;
		Xus_TN_MENU.bo_Update := TRUE;
		Xus_TN_SCREEN.by_Input_Exten_Code := BYTE#00;
	END_IF;
END_IF;

IF bo_Reset_Position = TRUE THEN
	bo_Reset_Position := FALSE;
	Xus_TN_MENU.in_X_SM_old := -1;
	Xus_TN_MENU.in_Y_SM_old := -1;
	Xus_TN_MENU.in_X_SM_new := -1;
	Xus_TN_MENU.in_Y_SM_new := -1;
END_IF;

(* POPUP-Menu updaten *)
IF (Xus_TN_MENU.in_State > INT#00) AND (Xus_TN_MENU.bo_Update = TRUE) THEN

	Xus_TN_MENU.bo_Update := FALSE; 

	in_ROW := Xus_TN_MENU.in_Y;
	in_COL := Xus_TN_MENU.in_X;

	(* Scrolloffset *)
	IF in_Scroll_Offset <> INT#00 THEN
		Xus_TN_MENU.in_Cur_Menu_Item := OSCAT_BASIC.INC2(Xus_TN_MENU.in_Cur_Menu_Item,in_Scroll_Offset,1,Xus_TN_MENU.in_Menu_E_Count);
		in_Scroll_Offset := INT#00;
	ELSE
		(* Item = 0 und kein Scrolloffset *)
		IF (Xus_TN_MENU.in_Cur_Menu_Item = INT#00) THEN
			Xus_TN_MENU.in_Cur_Menu_Item := INT#01;
		END_IF;
	END_IF;

	(* alle Menutext zeichnen *)
	FOR in_Count := INT#01 TO Xus_TN_MENU.in_Menu_E_Count DO;

		(* Zeichenfarbe bestimmen *)
		IF (in_Count = Xus_TN_MENU.in_Cur_Menu_Item) AND (Xus_TN_MENU.in_State > INT#01 ) THEN
			by_ATTR := Xus_TN_MENU.by_Attr_mF;

			Xus_TN_MENU.in_Y_SM_new := in_ROW + INT#01;
			Xus_TN_MENU.in_X_SM_new := in_COL;

		ELSE
			by_ATTR := Xus_TN_MENU.by_Attr_oF;
		END_IF;

		st_MENU_TITLE := ELEMENT_GET(SEP:=BYTE#35,POS:=in_Count - 1,ELEMENT:=st_MENU_BAR);

		in_TITLE_Length := LEN(st_MENU_TITLE) + INT#02;

		FB_TN_SC_WRITE_C(	Iin_Y := in_ROW,
							Iin_X := in_COL,
							Iby_ATTR := by_ATTR,
							Iin_LENGTH := in_TITLE_Length,
							Iin_OPTION := INT#02,
							Ist_STRING := st_MENU_TITLE,
							Xus_TN_SCREEN := Xus_TN_SCREEN);

		in_COL := in_COL + in_TITLE_Length;

	END_FOR;
END_IF;

IF Xus_TN_MENU.in_X_SM_new <> Xus_TN_MENU.in_X_SM_old THEN

	(* SubMenu ist aktiv -> beenden                                     *)
	IF us_TN_MENU_POPUP.bo_Activ = TRUE THEN
		us_TN_MENU_POPUP.bo_Destroy := TRUE;

		(* Sub-Menu bearbeiten *)
		FB_TN_INPUT_MENU_POPUP(	Xus_TN_MENU_POPUP := us_TN_MENU_POPUP,
								Xus_TN_SCREEN := Xus_TN_SCREEN);
	END_IF;

	IF us_TN_MENU_POPUP.bo_Activ = FALSE THEN
		(* Popup-Menu zu aktuellen Menu parametrieren und ausführen         *)
		in_Index := Xus_TN_MENU.in_Cur_Menu_Item;

		us_TN_MENU_POPUP.in_Y := Xus_TN_MENU.in_Y_SM_new;
		us_TN_MENU_POPUP.in_X := Xus_TN_MENU.in_X_SM_new;
		us_TN_MENU_POPUP.by_Attr_mF := Xus_TN_MENU.by_Attr_mF;
		us_TN_MENU_POPUP.by_Attr_oF := Xus_TN_MENU.by_Attr_oF;
		us_TN_MENU_POPUP.st_Menu_Text := ELEMENT_GET(SEP:=BYTE#37,POS:=in_Index,ELEMENT:=Xus_TN_MENU.st_MENU_TEXT);
		us_TN_MENU_POPUP.bo_Create := TRUE;

		Xus_TN_MENU.in_X_SM_old := Xus_TN_MENU.in_X_SM_new;
		Xus_TN_MENU.in_Y_SM_old := Xus_TN_MENU.in_Y_SM_new;

	END_IF;
END_IF;

(* Popup-Menu zyklisch aufrufen *)
FB_TN_INPUT_MENU_POPUP(	Xus_TN_MENU_POPUP := us_TN_MENU_POPUP,
						Xus_TN_SCREEN := Xus_TN_SCREEN);

(* aktuelles Item vom Popup-Menu kopieren *)
Xus_TN_MENU.in_Cur_Sub_Item := us_TN_MENU_POPUP.in_Cur_Item;

(* Destroy-Befehl *)
IF (Xus_TN_MENU.in_State = INT#01) THEN
	IF (Xus_TN_MENU.bo_Destroy = TRUE) THEN
		Xus_TN_MENU.in_State := INT#00;
		Xus_TN_MENU.bo_Destroy := FALSE;
		Xus_TN_MENU.in_Cur_Menu_Item := INT#00;
		Xus_TN_MENU.in_Cur_Sub_Item := INT#00;
	END_IF;
END_IF;

(* revision history
ks	06. apr. 2011	rev 1.1
	list_len und list_get durch element_count und element_get ersetzt

ks	10. mai. 2010	rev 1.0
	original version
*)

END_FUNCTION_BLOCK

// POUs/TELNET_VISION/TN_RECEIVE
FUNCTION_BLOCK TN_RECEIVE
VAR_IN_OUT
	R_BUF :	NETWORK_BUFFER;
	Xus_TN_SCREEN : us_TN_SCREEN;
END_VAR
VAR
	REQ_Size : UINT;
	REQ1 : BYTE;
	REQ2 : BYTE;
	REQ3 : BYTE;
END_VAR

(*
version 1.0		10. mai 2010
programmer		ks
tested by		ks

TN_RECEIVE empfängt Tastatureingaben vom Telnet Client und wertet diese aus
*)

(* Datenempfang auswertung *)
Xus_TN_SCREEN.by_Input_ASCII_Code := BYTE#00;
Xus_TN_SCREEN.by_Input_Exten_Code := BYTE#00;

IF R_BUF.SIZE > UINT#0 THEN
	(* empfangene Daten auswerten *)
	REQ_Size := R_BUF.SIZE;
	REQ1 := R_BUF.BUFFER[0];
	REQ2 := R_BUF.BUFFER[1];
	REQ3 := R_BUF.BUFFER[2];

	IF REQ1 = BYTE#27 AND REQ_Size >= UINT#3 THEN (* Escape *)
		IF REQ2 = BYTE#91 THEN (* Cursor code *)
			IF (REQ3 >= BYTE#65 AND REQ3 <= BYTE#68) OR (REQ3 = BYTE#72) OR (REQ3 = BYTE#75) THEN (* 65..68 = Cursor o,u,r,l / 72 = POS1 / 75 = ENDE *)
				Xus_TN_SCREEN.by_Input_Exten_Code := REQ3;
			END_IF;
		ELSIF REQ2 = BYTE#79 THEN (* Sondertasten F1/F2/F3/F4 *)
			IF REQ3 >= BYTE#80 AND REQ3 <= BYTE#83 THEN
				Xus_TN_SCREEN.by_Input_Exten_Code := REQ3;
			END_IF;
		END_IF;
	ELSIF REQ1 >= BYTE#32 AND REQ1 <= BYTE#126 THEN
		Xus_TN_SCREEN.by_Input_ASCII_Code := REQ1;
		Xus_TN_SCREEN.bo_Input_ASCII_IsNum := OSCAT_BASIC.ISC_NUM(REQ1); (* Auswertung auf Zahleneingabe *)
	ELSIF REQ1 = BYTE#8 OR REQ1 = BYTE#9 OR REQ1 = BYTE#13 OR REQ1 = BYTE#27 THEN (* prüfe auf Steuerzeichen 8=Backspace / 9=Tabulator / 13=Return / 27=Escape *)
		Xus_TN_SCREEN.by_Input_Exten_Code := REQ1;
	END_IF;

	(* Empfangsbuffer Datenlänge null eintragen (Telegramm zerstören *)
	R_BUF.SIZE := UINT#00;
END_IF;

(* revision history
ks	10. mai. 2010	rev 1.0
	original version
*)

END_FUNCTION_BLOCK

// POUs/TELNET_VISION/TN_SEND_ROWS
FUNCTION_BLOCK TN_SEND_ROWS
VAR_IN_OUT
	IP_C : IP_C;
	S_BUF : NETWORK_BUFFER;
	Xus_TN_SCREEN : us_TN_SCREEN;
END_VAR
VAR_INPUT
	S_BUF_SIZE : INT;
END_VAR
VAR
	in_Line_Count : INT;(*Zähler um max alle 24 Zeilen zu durchlaufen*)
	in_Col_Count : INT;
	in_Last_Row_Index : INT;
	bo_Break_Loop : BOOL;
	in_Row_Count : INT;
	in_Offset : INT;
	in_Write_Index : INT;
	in_Write_Index_Backup : INT;
	by_Cur_Color : BYTE;
	by_last_Color : BYTE;
	in_Write_Stop : INT;
END_VAR

(*
version 1.0		10. mai 2010
programmer		ks
tested by		ks

TN_SEND_ROWS prüft den Bildschirmspeicher auf änderungen, und sendet diese zeilenweise an den Telnet Client 
*)

(* Verbindung vorhanden und kein Datensenden aktiv *)
IF (IP_C.C_STATE < BYTE#127 OR S_BUF.SIZE > UINT#0) THEN
	RETURN; (* nein -> Baustein beenden *)
END_IF;

(* aktuellen Schreibindex laden *)
in_Write_Index := UINT_TO_INT(S_BUF.SIZE) - 1;

(* aktuellen Schreibindex zwischenspeichern *)
in_Write_Index_Backup := in_Write_Index;

(* positive Flanke Connect on *)
IF (IP_C.C_STATE = BYTE#254) OR (Xus_TN_SCREEN.bo_Clear_Screen) THEN

	(* Clear-Screen Meldung rücksetzen *)
	Xus_TN_SCREEN.bo_Clear_Screen := FALSE;

	(* alle Zeilen für Update markieren *)
	FOR in_Line_Count := INT#00 TO INT#23 DO
		Xus_TN_SCREEN.bya_Line_Update[in_Line_Count] := TRUE;
	END_FOR;

	(* ESC [0;30,40m  Reset Attributes + Black,Black *)
	in_Write_Index := in_Write_Index + INT#1;
	S_BUF.BUFFER[in_Write_Index] := BYTE#16#1B; (* ESC *)
	in_Write_Index := in_Write_Index + INT#1;
	S_BUF.BUFFER[in_Write_Index] := BYTE#16#5B; (* [ *)
	in_Write_Index := in_Write_Index + INT#1;
	S_BUF.BUFFER[in_Write_Index] := BYTE#16#30; (* 0 *)
	in_Write_Index := in_Write_Index + INT#1;
	S_BUF.BUFFER[in_Write_Index] := BYTE#16#3B; (* ; *)
	in_Write_Index := in_Write_Index + INT#1;
	S_BUF.BUFFER[in_Write_Index] := BYTE#16#33; (* 3 *)

	(* Einerstelle Farbe Foreground ausgeben *)
	in_Write_Index := in_Write_Index + INT#1;
	S_BUF.BUFFER[in_Write_Index] := (SHR(Xus_TN_SCREEN.by_Clear_Screen_Attr,4) OR BYTE#16#30);

	in_Write_Index := in_Write_Index + INT#1;
	S_BUF.BUFFER[in_Write_Index] := BYTE#16#3B; (* ; *)
	in_Write_Index := in_Write_Index + INT#1;
	S_BUF.BUFFER[in_Write_Index] := BYTE#16#34; (* 4 *)

	(* Einerstelle Farbe Background ausgeben *)
	in_Write_Index := in_Write_Index + INT#1;
	S_BUF.BUFFER[in_Write_Index] := ((Xus_TN_SCREEN.by_Clear_Screen_Attr AND BYTE#16#07) OR BYTE#16#30);

	in_Write_Index := in_Write_Index + INT#1;
	S_BUF.BUFFER[in_Write_Index] := BYTE#16#6D; (* m *)

	(* ESC[2J Clear screen and home cursor *)
	in_Write_Index := in_Write_Index + INT#1;
	S_BUF.BUFFER[in_Write_Index] := BYTE#16#1B; (* ESC *)
	in_Write_Index := in_Write_Index + INT#1;
	S_BUF.BUFFER[in_Write_Index] := BYTE#16#5B; (* [ *)
	in_Write_Index := in_Write_Index + INT#1;
	S_BUF.BUFFER[in_Write_Index] := BYTE#16#32; (* 2 *)
	in_Write_Index := in_Write_Index + INT#1;
	S_BUF.BUFFER[in_Write_Index] := BYTE#16#4A; (* J *)

	(* ESC [?7l Off *)
	in_Write_Index := in_Write_Index + INT#1;
	S_BUF.BUFFER[in_Write_Index] := BYTE#16#1B; (* ESC *)
	in_Write_Index := in_Write_Index + INT#1;
	S_BUF.BUFFER[in_Write_Index] := BYTE#16#5B; (* [ *)
	in_Write_Index := in_Write_Index + INT#1;
	S_BUF.BUFFER[in_Write_Index] := BYTE#16#3F; (* ? *)
	in_Write_Index := in_Write_Index + INT#1;
	S_BUF.BUFFER[in_Write_Index] := BYTE#16#37; (* 7 *)
	in_Write_Index := in_Write_Index + INT#1;
	S_BUF.BUFFER[in_Write_Index] := BYTE#16#6C; (* l *)

END_IF;

in_Last_Row_Index := INT#0;
bo_Break_Loop := FALSE;
in_Write_Stop := S_BUF_SIZE - 20;

(* alle Zeilen durchlaufen *)
FOR in_Line_Count := 0 TO 23 DO

	in_Offset := in_Row_Count * INT#80;

	(* prüfen ob Update einer Zeile notwendig ist bzw. nach Reconnect *)
	IF (Xus_TN_SCREEN.bya_Line_Update[in_Row_Count] = TRUE) THEN

		(* Schreib-Cursor positionieren *)
		in_Write_Index := in_Write_Index + INT#1;
		S_BUF.BUFFER[in_Write_Index] := BYTE#16#1B; (* ESC *)
		in_Write_Index := in_Write_Index + INT#1;
		S_BUF.BUFFER[in_Write_Index] := BYTE#16#5B; (* [ *)

		(* Zehnerstelle Zeilennummer ausgeben *)
		in_Write_Index := in_Write_Index + INT#1;
		S_BUF.BUFFER[in_Write_Index] :=
		SHR(OSCAT_BASIC.INT_TO_BCDC(in_Row_Count + INT#1),INT#4) OR BYTE#16#30;

		(* Einerstelle Zeilennummer ausgeben *)
		in_Write_Index := in_Write_Index + INT#1;
		S_BUF.BUFFER[in_Write_Index] :=
		(OSCAT_BASIC.INT_TO_BCDC(in_Row_Count + INT#1) AND BYTE#16#0F) OR BYTE#16#30;

		in_Write_Index := in_Write_Index + INT#1;
		S_BUF.BUFFER[in_Write_Index] := BYTE#16#3B; (* ; *)
		in_Write_Index := in_Write_Index + INT#1;
		S_BUF.BUFFER[in_Write_Index] := BYTE#16#31; (* 1 *)
		in_Write_Index := in_Write_Index + INT#1;
		S_BUF.BUFFER[in_Write_Index] := BYTE#16#48; (* H *)

		(* alle Spalten einer Zeile durchlaufen *)
		FOR in_Col_Count := 0 TO 79 DO

			(* aktuelle Farbe bestimmen *)
			by_Cur_Color := Xus_TN_SCREEN.bya_COLOR[in_Offset];
			IF (by_Cur_Color <> by_last_Color) OR (in_Col_Count = INT#00) THEN

				(* Farbeinstellung: ANSI-Sequenz ESC[X;Y;Zm ausgeben *)
				in_Write_Index := in_Write_Index + INT#1;
				S_BUF.BUFFER[in_Write_Index] := BYTE#16#1B; (* ESC *)

				in_Write_Index := in_Write_Index + INT#1;
				S_BUF.BUFFER[in_Write_Index] := BYTE#16#5B; (* [ *)

				(* Farbeinstellung: dunkel oder Hell und blinken bestimmen *)

					IF (((by_Cur_Color AND BYTE#2#10001000) XOR (by_last_Color AND BYTE#2#10001000)) <> BYTE#00) OR (in_Col_Count = 0) THEN

						in_Write_Index := in_Write_Index + INT#1;
						S_BUF.BUFFER[in_Write_Index] := BYTE#16#30; (* 0 *)
						in_Write_Index := in_Write_Index + INT#1;
						S_BUF.BUFFER[in_Write_Index] := BYTE#16#3B; (* ; *)

						(* keine dunklen Farben gewünscht -> dann Bold & Bright *)
						IF (by_Cur_Color AND BYTE#2#00001000) = BYTE#2#00000000 THEN

							(* auf Bold & Btight Farben umstellen *)
							in_Write_Index := in_Write_Index + INT#1;
							S_BUF.BUFFER[in_Write_Index] := BYTE#16#31; (* 1 *) 
							in_Write_Index := in_Write_Index + INT#1;
							S_BUF.BUFFER[in_Write_Index] := BYTE#16#3B; (* ; *)

						END_IF;

						(* blinkenden Farben gewünscht *)
						IF (by_Cur_Color AND BYTE#2#10000000) = BYTE#2#10000000 THEN 

							(* auf Bold & Bright Farben umstellen *)
							in_Write_Index := in_Write_Index + INT#1;
							S_BUF.BUFFER[in_Write_Index] := BYTE#16#35; (* 5 *) 
							in_Write_Index := in_Write_Index + INT#1;
							S_BUF.BUFFER[in_Write_Index] := BYTE#16#3B; (* ; *)

						END_IF;

					END_IF;

					(* Zehnerstelle Farbe Foreground ausgeben *)
					in_Write_Index := in_Write_Index + INT#1;
					S_BUF.BUFFER[in_Write_Index] := BYTE#16#33; (* 3 *)

					(* Einerstelle Farbe Foreground ausgeben *)
					in_Write_Index := in_Write_Index + INT#1;
					S_BUF.BUFFER[in_Write_Index] := ((SHR(by_Cur_Color,4) AND BYTE#2#00000111) OR BYTE#16#30);

					in_Write_Index := in_Write_Index + INT#1;
					S_BUF.BUFFER[in_Write_Index] := BYTE#16#3B; (* ; *)

					(* Zehnerstelle Farbe Background ausgeben *)
					in_Write_Index := in_Write_Index + INT#1;
					S_BUF.BUFFER[in_Write_Index] := BYTE#16#34; (* 4 *)

					(* Einerstelle Farbe Background ausgeben *)
					in_Write_Index := in_Write_Index + INT#1;
					S_BUF.BUFFER[in_Write_Index] := ((by_Cur_Color AND BYTE#2#00000111) OR BYTE#16#30); 

					in_Write_Index := in_Write_Index + INT#1;
					S_BUF.BUFFER[in_Write_Index] := BYTE#16#6D; (* m *)

					(* neue Farbe als letzt verwendete speichern *)
					by_last_Color := by_Cur_Color;

				END_IF;

				(* Buffer Ende vorzeitig erreicht -> Ende *)
				IF (in_Write_Index > in_Write_Stop) THEN

					bo_Break_Loop := TRUE;
					EXIT;

				END_IF;

				(* ein TEXT-Zeichen von Screenbuffer in den Sendebuffer übertragen *)
				in_Write_Index := in_Write_Index + INT#1;
				S_BUF.BUFFER[in_Write_Index] := Xus_TN_SCREEN.bya_CHAR[in_Offset];

				(* nächste Spalte anwählen *)
				in_Offset := in_Offset + INT#01;
			END_FOR;

			IF (bo_Break_Loop = TRUE) THEN;

				(* Buffer Ende vorzeitig erreicht -> nur bis zur letzten kompletten Zeile uebertragen *)
				in_Write_Index := in_Last_Row_Index;

				EXIT;
			END_IF;

			(* Buffer ist noch nicht voll -> neue Zeile ubernehmen *)
			in_Last_Row_Index := in_Write_Index;
			Xus_TN_SCREEN.bya_Line_Update[in_Row_Count] := FALSE;

		END_IF;

		(* naechste Zeile adressieren *)
		in_Row_Count := in_Row_Count + INT#01;

		(* ab letzter Zeile wieder von vorne beginnen *)
		IF (in_Row_Count > INT#23) THEN
			in_Row_Count := INT#00;
		END_IF;
		(*-----------------------------------------------*)


	END_FOR;

	(* wenn in einen Update-Zyklus alle Zeilen auf einmal geschafft wurden *)
	(* wird der Row_Count auf ersten Zeile gestellt *)
	(* soll das hässliche Grafikflackern verhindern *)
	(* ansonsten wird bei der letzen Zeile weitergemacht *)
	IF (bo_Break_Loop = FALSE) THEN
		in_Row_Count := INT#00;
	END_IF;

	(* Edit-Cursor positionieren *)
	IF (in_Write_Index <> in_Write_Index_Backup) THEN

		in_Write_Index := in_Write_Index + INT#1;
		S_BUF.BUFFER[in_Write_Index] := BYTE#16#1B; (* ESC *)
		in_Write_Index := in_Write_Index + INT#1;
		S_BUF.BUFFER[in_Write_Index] := BYTE#16#5B; (* [ *)

		(* Zehnerstelle Zeilennummer ausgeben *)
		in_Write_Index := in_Write_Index + INT#1;
		S_BUF.BUFFER[in_Write_Index] := SHR(OSCAT_BASIC.INT_TO_BCDC(Xus_TN_SCREEN.in_Cursor_Y + 1),INT#4) OR BYTE#16#30;

		(* Einerstelle Zeilennummer ausgeben *)
		in_Write_Index := in_Write_Index + INT#1;
		S_BUF.BUFFER[in_Write_Index] := (OSCAT_BASIC.INT_TO_BCDC(Xus_TN_SCREEN.in_Cursor_Y + 1) AND BYTE#16#0F) OR BYTE#16#30;

		in_Write_Index := in_Write_Index + INT#1;
		S_BUF.BUFFER[in_Write_Index] := BYTE#16#3B; (* ; *)

		(* Zehnerstelle Spaltenummer ausgeben *)
		in_Write_Index := in_Write_Index + INT#1;
		S_BUF.BUFFER[in_Write_Index] := SHR(OSCAT_BASIC.INT_TO_BCDC(Xus_TN_SCREEN.in_Cursor_X + 1),INT#4) OR BYTE#16#30;

		(* Einerstelle Spaltennummer ausgeben *)
		in_Write_Index := in_Write_Index + INT#1;
		S_BUF.BUFFER[in_Write_Index] := (OSCAT_BASIC.INT_TO_BCDC(Xus_TN_SCREEN.in_Cursor_X + 1) AND BYTE#16#0F) OR BYTE#16#30;

		in_Write_Index := in_Write_Index + INT#1;
		S_BUF.BUFFER[in_Write_Index] := BYTE#16#48; (* H *)

END_IF;

(* aktuellen Schreibindex speichern -> Senden anstossen *)
S_BUF.SIZE := INT_TO_UINT(in_Write_Index + 1);

(* revision history
ks	10. mai. 2010	rev 1.0
	original version
*)

END_FUNCTION_BLOCK

// POUs/TELNET_VISION/TN_SC_READ_ATTR
FUNCTION_BLOCK TN_SC_READ_ATTR
VAR
	in_Offset : INT;
END_VAR
VAR_INPUT
	Iin_Y : INT;
	Iin_X : INT;
END_VAR
VAR_OUTPUT
	Oby_ATTR : BYTE;
END_VAR
VAR_IN_OUT
	Xus_TN_SCREEN : us_TN_SCREEN;
END_VAR

(*
version 1.0		10. mai 2010
programmer		ks
tested by		ks

TN_SC_READ_ATTR gibt den Farbcode einer Koordinate vom Bildschirm aus

*)

IF TN_SC_XY_ERROR(Iin_X,Iin_Y) THEN RETURN; END_IF;
in_Offset := (Iin_Y * 80) + Iin_X;
Oby_ATTR := Xus_TN_SCREEN.bya_COLOR[in_Offset]; (* Attribute auslesen *)

(* revision history
ks	10. mai. 2010	rev 1.0
	original version
*)

END_FUNCTION_BLOCK

// POUs/TELNET_VISION/TN_SC_READ_CHAR
FUNCTION_BLOCK TN_SC_READ_CHAR
VAR
	in_Offset : INT;
END_VAR
VAR_INPUT
	Iin_Y : INT;
	Iin_X : INT;
END_VAR
VAR_OUTPUT
	Oby_CHAR : BYTE;
END_VAR
VAR_IN_OUT
	Xus_TN_SCREEN : us_TN_SCREEN;
END_VAR

(*
version 1.0		10. mai 2010
programmer		ks
tested by		ks

TN_SC_READ_CHAR gibt das Zeichen einer Koordinate vom Bildschirm aus
*)

IF TN_SC_XY_ERROR(Iin_X,Iin_Y) THEN RETURN; END_IF;
in_Offset := (Iin_Y * 80) + Iin_X;
Oby_CHAR := Xus_TN_SCREEN.bya_CHAR[in_Offset]; (* Charakter auslesen *)

(* revision history
ks	10. mai. 2010	rev 1.0
	original version
*)

END_FUNCTION_BLOCK

// POUs/TELNET_VISION/TN_SC_VIEWPORT
FUNCTION_BLOCK TN_SC_VIEWPORT
VAR
	FB_TN_SC_WRITE : TN_SC_WRITE;
	FB_TON : TON;
END_VAR
VAR
	in_index : INT;
	in_Color : INT;
	by_Attr : BYTE;
	in_count : INT;
END_VAR
VAR_IN_OUT
	Xus_LOG_VIEWPORT : us_LOG_VIEWPORT;
	Xus_LOG_CONTROL : LOG_CONTROL;
	Xus_TN_SCREEN : us_TN_SCREEN;
END_VAR
VAR_INPUT
	Iin_X : INT;
	Iin_Y : INT;
	Iin_Width : INT;
	Idw_ATTR_1 : DWORD;
	Idw_ATTR_2 : DWORD;
	Iti_TIME : TIME;
END_VAR

(*
version 1.0		10. mai 2010
programmer		ks
tested by		ks

TN_SC_VIEWPORT verwaltet und zeichnet einen rechteckigen Bereich in dem der Log-buffer angezeigt wird
*)

(* LOG-Messages ausgeben *)

IF Xus_LOG_VIEWPORT.UPDATE AND FB_TON.Q THEN (* Update gewünscht und Verzögerungszeit abgelaufen *)
	Xus_LOG_VIEWPORT.UPDATE := FALSE;
	FOR in_count := 1 TO Xus_LOG_VIEWPORT.COUNT DO (* Alle Viewport-Zeilen abarbeiten *)
		in_index := Xus_LOG_VIEWPORT.LINE_ARRAY[in_count];
		(* Farbe aus den Option-Parameter auslesen >0,Level,Back,Front< *)
		in_Color := DWORD_TO_INT(Xus_LOG_CONTROL.MSG_OPTION[in_index] AND DWORD#2#1111);

		CASE in_Color OF
		0..3: by_Attr := OSCAT_BASIC.BYTE_OF_DWORD(Idw_ATTR_1,INT_TO_BYTE(in_Color));
		4..7: by_Attr := OSCAT_BASIC.BYTE_OF_DWORD(Idw_ATTR_2,INT_TO_BYTE(in_Color));
		ELSE
			by_Attr := OSCAT_BASIC.BYTE_OF_DWORD(Idw_ATTR_1,BYTE#0);
		END_CASE;

		(* Message (Text + Farbe) ausgeben *)
		FB_TN_SC_WRITE(	Iin_Y := Iin_Y + in_count - INT#01,
						Iin_X := Iin_X,
						Iby_ATTR := by_Attr,
						Ist_STRING := OSCAT_BASIC.FIX(str := Xus_LOG_CONTROL.MSG[in_index], L := Iin_Width, C := BYTE#32, M := INT#00), (* String rechts ergänzen bzw. kürzen *)
						Xus_TN_SCREEN := Xus_TN_SCREEN);

	END_FOR;

	(* Timer stoppen/rücksetzen *)
	FB_TON.IN := FALSE;
	FB_TON.PT := Iti_TIME;
	FB_TON();

END_IF;

(* Update-Zeitverzoegerung *)
FB_TON.IN := TRUE;
FB_TON.PT := Iti_TIME;
FB_TON();

(* revision history
ks	10. mai. 2010	rev 1.0
	original version
*)

END_FUNCTION_BLOCK

// POUs/TELNET_VISION/TN_SC_WRITE_ATTR
FUNCTION_BLOCK TN_SC_WRITE_ATTR
VAR
	in_Offset : INT;
END_VAR
VAR_INPUT
	Iin_Y : INT;
	Iin_X : INT;
	Iby_ATTR : BYTE;
END_VAR
VAR_IN_OUT
	Xus_TN_SCREEN : us_TN_SCREEN;
END_VAR

(*
version 1.0		10. mai 2010
programmer		ks
tested by		ks

TN_SC_WRITE_ATTR ändert an der angegebenen Koordinate den Farbcode
*)

IF TN_SC_XY_ERROR(Iin_X,Iin_Y) THEN RETURN; END_IF;
in_Offset := (Iin_Y * 80) + Iin_X;
Xus_TN_SCREEN.bya_COLOR[in_Offset] := Iby_ATTR; (* Attribute schreiben *)

(* revision history
ks	10. mai. 2010	rev 1.0
	original version
*)

END_FUNCTION_BLOCK

// POUs/TELNET_VISION/TN_SC_WRITE_CHAR
FUNCTION_BLOCK TN_SC_WRITE_CHAR
VAR
	in_Offset : INT;
END_VAR
VAR_INPUT
	Iin_Y : INT;
	Iin_X : INT;
	Iby_CHAR : BYTE;
END_VAR
VAR_IN_OUT
	Xus_TN_SCREEN : us_TN_SCREEN;
END_VAR

(*
version 1.0		10. mai 2010
programmer		ks
tested by		ks

TN_SC_WRITE_CHAR schreibt ein einzelnes Zeichen an die angegebenen Koordinate ohne den vorhandenen Farbcode zu ändern 
*)

IF TN_SC_XY_ERROR(Iin_X,Iin_Y) THEN RETURN; END_IF;
in_Offset := (Iin_Y * 80) + Iin_X;
Xus_TN_SCREEN.bya_CHAR[in_Offset] := Iby_CHAR; (* Charakter schreiben *)

(* revision history
ks	10. mai. 2010	rev 1.0
	original version
*)

END_FUNCTION_BLOCK

// POUs/TELNET_VISION/TN_SC_WRITE_EOS
FUNCTION_BLOCK TN_SC_WRITE_EOS
VAR
	TN_SC_WRITE : TN_SC_WRITE;
END_VAR
VAR_INPUT
	Iby_ATTR : BYTE;
	Ist_STRING : STRING;
END_VAR
VAR_IN_OUT
	Xus_TN_SCREEN : us_TN_SCREEN;
END_VAR

(*
version 1.0		10. mai 2010
programmer		ks
tested by		ks

TN_SC_WRITE_EOS schreibt einem Text an das Ende des zuletzt geschreibene Texts 
*)

TN_SC_WRITE(Iin_Y := Xus_TN_SCREEN.in_EOS_Offset / 80, (* aktuelle Zeile ausrechnen *)
			Iin_X := Xus_TN_SCREEN.in_EOS_Offset MOD 80, (* aktuelle Spalte ausrechnen *)
			Iby_ATTR := Iby_ATTR,
			Ist_STRING := Ist_STRING,
			Xus_TN_SCREEN := Xus_TN_SCREEN);

(* revision history
ks	10. mai. 2010	rev 1.0
	original version
*)

END_FUNCTION_BLOCK

// POUs/DEMO/TN_VISION_DEMO_1
PROGRAM TN_VISION_DEMO_1
VAR
	FB_TN_FRAMEWORK : TN_FRAMEWORK;
	FB_LOG_MESSAGE : LOG_MSG;
	FB_LOG_VIEWPORT : LOG_VIEWPORT;
	FB_TN_SC_LINE : TN_SC_LINE;
	FB_TN_SC_FILL : TN_SC_FILL;
	FB_TN_SC_WRITE_C : TN_SC_WRITE_C;
	FB_TN_SC_BOX : TN_SC_BOX;
	FB_TN_SC_ADD_SHADOW : TN_SC_ADD_SHADOW;
	FB_TN_SC_WRITE : TN_SC_WRITE;
	FB_TN_SC_VIEWPORT : TN_SC_VIEWPORT;
	Xus_TN_MENU : us_TN_MENU;
	Xus_TN_INPUT_CONTROL : us_TN_INPUT_CONTROL;
	Xus_TN_SCREEN : us_TN_SCREEN;
	us_LOG_VIEWPORT : us_LOG_VIEWPORT;
	S_BUF : NETWORK_BUFFER;
	R_BUF : NETWORK_BUFFER;
	IP_C : IP_C;
	Gst_SysLog_Command : STRING;
	in_index : INT;
END_VAR

FB_TN_FRAMEWORK(
					us_TN_INPUT_CONTROL := Xus_TN_INPUT_CONTROL ,
					us_TN_SCREEN := Xus_TN_SCREEN ,
					us_TN_MENU := Xus_TN_MENU ,
					S_BUF := S_BUF ,
					R_BUF:= R_BUF ,
					IP_C:= IP_C ,
					PORT := WORD#0
					 );

(* Modaler Dialog aktiv ? *)
IF (Xus_TN_SCREEN.bo_Modal_Dialog = TRUE) THEN RETURN; END_IF;

IF Xus_TN_MENU.in_Menu_Selected > 0 THEN

	CASE Xus_TN_MENU.in_Menu_Selected OF

	41: (* Seite LOGIN aufrufen *)
		Xus_TN_SCREEN.in_Page_Number := INT#00;
		(* Gedächtnis löschen *)
		Xus_TN_MENU.bo_Destroy := TRUE;

	END_CASE;

	(* Echo Menu-Auswahl *)
	Gst_SysLog_Command := CONCAT('MENU_SELECT: ',INT_TO_STRING(Xus_TN_MENU.in_Menu_Selected));

	(* Menu-Auswahl löschen *)
	Xus_TN_MENU.in_Menu_Selected := 0;

END_IF;

(* Initialisierung der Daten und Strukturen *)
IF (Xus_TN_SCREEN.in_Page_Number = INT#00 ) THEN
	Xus_TN_SCREEN.in_Page_Number := INT#01;

	(* Clear-Screen (Farbe setzen + Display löschen) *)
	Xus_TN_SCREEN.by_Clear_Screen_Attr := BYTE#16#00;
	Xus_TN_SCREEN.bo_Clear_Screen := TRUE;

	(* Screen initialisieren (mit Leerzeichen füllen) *)
	FB_TN_SC_FILL(	Iin_X1 := INT#00,
					Iin_Y1 := INT#00,
					Iin_X2 := INT#79,
					Iin_Y2 := INT#23,
					Iby_CHAR := BYTE#179,
					Iby_Attr := BYTE#16#76,
					Xus_TN_SCREEN := Xus_TN_SCREEN);

	(* Titlezeile zeichnen *)
	FB_TN_SC_FILL(	Iin_X1 := INT#00,
					Iin_Y1 := INT#00,
					Iin_X2 := INT#79,
					Iin_Y2 := INT#00,
					Iby_CHAR := BYTE#32,
					Iby_Attr := BYTE#16#07,
					Xus_TN_SCREEN := Xus_TN_SCREEN);

	(* Title zeichnen *)
	FB_TN_SC_WRITE(	Iin_X := INT#00,
					Iin_Y := INT#00,
					Iby_ATTR := BYTE#16#77,
					Ist_STRING := ' TELNET-VISION BIOS v1.0',
					Xus_TN_SCREEN := Xus_TN_SCREEN);

	(* Fusszeile zeichnen *)
	FB_TN_SC_FILL(	Iin_X1 := INT#00,
					Iin_Y1 := INT#23,
					Iin_X2 := INT#79,
					Iin_Y2 := INT#23,
					Iby_CHAR := BYTE#32,
					Iby_Attr := BYTE#16#37,
					Xus_TN_SCREEN := Xus_TN_SCREEN);

	(* Rahmen für Viewport zeichnen *)
	FB_TN_SC_BOX(	Iin_X1 := INT#03,
					Iin_Y1 := INT#03,
					Iin_X2 := INT#75,
					Iin_Y2 := INT#19,
					Iby_FILL := BYTE#16#20, (* Füllung *)
					Iin_BORDER := INT#02, (* Double-Line Border *)
					Iby_ATTR := BYTE#16#74, (* Weiss , Blau *)
					Xus_TN_SCREEN := Xus_TN_SCREEN);

	(* Shadow für Rahmen von Viewport zeichnen *)
	FB_TN_SC_ADD_SHADOW(	Iin_X1 := INT#04,
							Iin_Y1 := INT#04,
							Iin_X2 := INT#76,
							Iin_Y2 := INT#20,
							Iin_OPTION := INT#00,
							Xus_TN_SCREEN := Xus_TN_SCREEN);

	(* Title Viewport zeichnen *)
	FB_TN_SC_WRITE(	Iin_X := INT#31,
					Iin_Y := INT#03,
					Iby_ATTR := BYTE#16#74,
					Ist_STRING := '[ LOGIN-DIALOG ]',
					Xus_TN_SCREEN := Xus_TN_SCREEN);

	(* LOGO Zeilen zeichnen *)
	FOR in_index := 5 TO 16 DO

		CASE in_index OF

		05: FB_TN_SC_WRITE.Ist_STRING := 'ÛÛÛÛÛÛÛÛ» ÛÛÛÛÛÛÛ» ÛÛ»      ÛÛÛ»   ÛÛ» ÛÛÛÛÛÛÛ» ÛÛÛÛÛÛÛÛ»';
		06: FB_TN_SC_WRITE.Ist_STRING := 'ÈÍÍÛÛÉÍÍ¼ ÛÛÉÍÍÍÍ¼ ÛÛº      ÛÛÛÛ»  ÛÛº ÛÛÉÍÍÍÍ¼ ÈÍÍÛÛÉÍÍ¼';
		07: FB_TN_SC_WRITE.Ist_STRING := '   ÛÛº    ÛÛÛÛÛ»   ÛÛº      ÛÛÉÛÛ» ÛÛº ÛÛÛÛÛ»      ÛÛº';
		08: FB_TN_SC_WRITE.Ist_STRING := '   ÛÛº    ÛÛÉÍÍ¼   ÛÛº      ÛÛºÈÛÛ»ÛÛº ÛÛÉÍÍ¼      ÛÛº';
		09: FB_TN_SC_WRITE.Ist_STRING := '   ÛÛº    ÛÛÛÛÛÛÛ» ÛÛÛÛÛÛÛ» ÛÛº ÈÛÛÛÛº ÛÛÛÛÛÛÛ»    ÛÛº';
		10: FB_TN_SC_WRITE.Ist_STRING := '   ÈÍ¼    ÈÍÍÍÍÍÍ¼ ÈÍÍÍÍÍÍ¼ ÈÍ¼  ÈÍÍÍ¼ ÈÍÍÍÍÍÍ¼    ÈÍ¼';
		11: FB_TN_SC_WRITE.Ist_STRING := '     ÛÛ»   ÛÛ» ÛÛ» ÛÛÛÛÛÛÛ» ÛÛ»  ÛÛÛÛÛÛ»  ÛÛÛ»   ÛÛ»';
		12: FB_TN_SC_WRITE.Ist_STRING := '     ÛÛº   ÛÛº ÛÛº ÛÛÉÍÍÍÍ¼ ÛÛº ÛÛÉÍÍÍÛÛ» ÛÛÛÛ»  ÛÛº';
		13: FB_TN_SC_WRITE.Ist_STRING := '     ÛÛº   ÛÛº ÛÛº ÛÛÛÛÛÛÛ» ÛÛº ÛÛº   ÛÛº ÛÛÉÛÛ» ÛÛº';
		14: FB_TN_SC_WRITE.Ist_STRING := '     ÈÛÛ» ÛÛÉ¼ ÛÛº ÈÍÍÍÍÛÛº ÛÛº ÛÛº   ÛÛº ÛÛºÈÛÛ»ÛÛº';
		15: FB_TN_SC_WRITE.Ist_STRING := '      ÈÛÛÛÛÉ¼  ÛÛº ÛÛÛÛÛÛÛº ÛÛº ÈÛÛÛÛÛÛÉ¼ ÛÛº ÈÛÛÛÛº';
		16: FB_TN_SC_WRITE.Ist_STRING := '       ÈÍÍÍ¼   ÈÍ¼ ÈÍÍÍÍÍÍ¼ ÈÍ¼  ÈÍÍÍÍÍ¼  ÈÍ¼  ÈÍÍÍ¼';

		END_CASE;

		FB_TN_SC_WRITE(	Iin_Y := in_index,
						Iin_X := INT#11,
						Iby_ATTR := BYTE#16#34,
						Xus_TN_SCREEN := Xus_TN_SCREEN);
	END_FOR;

	(* Trennlinie zeichnen *)
	FB_TN_SC_LINE(	Iin_X1 := INT#03,
					Iin_Y1 := INT#17,
					Iin_X2 := INT#75,
					Iin_Y2 := INT#17,
					Iby_ATTR := BYTE#16#74,
					Iby_BORDER := BYTE#02,
					Xus_TN_SCREEN := Xus_TN_SCREEN);

	(* Alle Input-Controls initialisieren *)

	Xus_TN_INPUT_CONTROL.bo_Enable := FALSE;

	(* Initialisierung der Eingabe-Zeile *)
	Xus_TN_INPUT_CONTROL.usa_TN_INPUT_CONTROL_DATA[1].in_Type := INT#01;
	Xus_TN_INPUT_CONTROL.usa_TN_INPUT_CONTROL_DATA[1].in_Y := INT#18;
	Xus_TN_INPUT_CONTROL.usa_TN_INPUT_CONTROL_DATA[1].in_X := INT#49;
	Xus_TN_INPUT_CONTROL.usa_TN_INPUT_CONTROL_DATA[1].by_Attr_mF := BYTE#16#17;
	Xus_TN_INPUT_CONTROL.usa_TN_INPUT_CONTROL_DATA[1].by_Attr_oF := BYTE#16#47;
	Xus_TN_INPUT_CONTROL.usa_TN_INPUT_CONTROL_DATA[1].in_Cursor_Pos := INT#0;
	Xus_TN_INPUT_CONTROL.usa_TN_INPUT_CONTROL_DATA[1].bo_Input_Only_Num := FALSE;
	Xus_TN_INPUT_CONTROL.usa_TN_INPUT_CONTROL_DATA[1].bo_Input_Hidden := TRUE;
	Xus_TN_INPUT_CONTROL.usa_TN_INPUT_CONTROL_DATA[1].st_Input_Mask := '                ';
	Xus_TN_INPUT_CONTROL.usa_TN_INPUT_CONTROL_DATA[1].st_Input_Data := Xus_TN_INPUT_CONTROL.usa_TN_INPUT_CONTROL_DATA[1].st_Input_Mask;
	Xus_TN_INPUT_CONTROL.usa_TN_INPUT_CONTROL_DATA[1].st_Input_ToolTip := ' enter password | press enter to login     |';
	Xus_TN_INPUT_CONTROL.usa_TN_INPUT_CONTROL_DATA[1].in_Input_Option := INT#00;
	Xus_TN_INPUT_CONTROL.usa_TN_INPUT_CONTROL_DATA[1].in_Title_Y_Offset := INT#00;
	Xus_TN_INPUT_CONTROL.usa_TN_INPUT_CONTROL_DATA[1].in_Title_X_Offset := -12;
	Xus_TN_INPUT_CONTROL.usa_TN_INPUT_CONTROL_DATA[1].by_Title_Attr := BYTE#16#34;
	Xus_TN_INPUT_CONTROL.usa_TN_INPUT_CONTROL_DATA[1].st_Title_String := 'password:  [                ]';

	(* Initialisierung Selection Text *)
	Xus_TN_INPUT_CONTROL.usa_TN_INPUT_CONTROL_DATA[2].in_Type := INT#03;
	Xus_TN_INPUT_CONTROL.usa_TN_INPUT_CONTROL_DATA[2].in_Y := INT#18;
	Xus_TN_INPUT_CONTROL.usa_TN_INPUT_CONTROL_DATA[2].in_X := INT#18;
	Xus_TN_INPUT_CONTROL.usa_TN_INPUT_CONTROL_DATA[2].by_Attr_mF := BYTE#16#17;
	Xus_TN_INPUT_CONTROL.usa_TN_INPUT_CONTROL_DATA[2].by_Attr_oF := BYTE#16#47;
	Xus_TN_INPUT_CONTROL.usa_TN_INPUT_CONTROL_DATA[2].st_Input_ToolTip := ' select user       | press enter to select |';
	Xus_TN_INPUT_CONTROL.usa_TN_INPUT_CONTROL_DATA[2].in_Input_Option := INT#00;
	Xus_TN_INPUT_CONTROL.usa_TN_INPUT_CONTROL_DATA[2].in_Title_Y_Offset := INT#00;
	Xus_TN_INPUT_CONTROL.usa_TN_INPUT_CONTROL_DATA[2].in_Title_X_Offset := INT#00;
	Xus_TN_INPUT_CONTROL.usa_TN_INPUT_CONTROL_DATA[2].by_Title_Attr := BYTE#16#34;
	Xus_TN_INPUT_CONTROL.usa_TN_INPUT_CONTROL_DATA[2].st_Title_String := ' user ';
	Xus_TN_INPUT_CONTROL.usa_TN_INPUT_CONTROL_DATA[2].st_Input_Mask := '           ';
	Xus_TN_INPUT_CONTROL.usa_TN_INPUT_CONTROL_DATA[2].st_Input_Data := 'admin#guest#maintenance';

	(* Control-Tool-Tip *)
	Xus_TN_INPUT_CONTROL.in_ToolTip_Y := INT#23;
	Xus_TN_INPUT_CONTROL.in_ToolTip_X := INT#00;
	Xus_TN_INPUT_CONTROL.by_ToolTip_Attr := BYTE#16#37;
	Xus_TN_INPUT_CONTROL.in_ToolTip_Size := INT#80;

	(* Control-Verwaltung initialisieren *)
	Xus_TN_INPUT_CONTROL.in_Count := INT#02;
	Xus_TN_INPUT_CONTROL.bo_Enable := TRUE;
	Xus_TN_INPUT_CONTROL.bo_Reset_Fokus := TRUE;

END_IF;

IF (Xus_TN_SCREEN.in_Page_Number = INT#01) THEN
	(* eingegebenen String übernehmen *)
	IF Xus_TN_INPUT_CONTROL.usa_TN_INPUT_CONTROL_DATA[1].bo_Input_Entered = TRUE THEN

		Xus_TN_INPUT_CONTROL.usa_TN_INPUT_CONTROL_DATA[1].bo_Input_Entered := FALSE;
		Xus_TN_INPUT_CONTROL.usa_TN_INPUT_CONTROL_DATA[1].st_Input_String :=
			OSCAT_BASIC.LOWERCASE(str:=Xus_TN_INPUT_CONTROL.usa_TN_INPUT_CONTROL_DATA[1].st_Input_String);

		IF Xus_TN_INPUT_CONTROL.usa_TN_INPUT_CONTROL_DATA[1].st_Input_String = 'oscat' THEN
			Xus_TN_SCREEN.in_Page_Number := INT#10;

			Gst_SysLog_Command := CONCAT('LOGON: USER-',Xus_TN_INPUT_CONTROL.usa_TN_INPUT_CONTROL_DATA[2].st_Input_String);

		ELSE
			FB_TN_SC_WRITE_C(	Iin_X := Xus_TN_INPUT_CONTROL.in_ToolTip_X,
								Iin_Y := Xus_TN_INPUT_CONTROL.in_ToolTip_Y,
								Iby_ATTR := BYTE#16#F1,
								Iin_OPTION := INT#02, (* Center-String *)
								Iin_LENGTH := Xus_TN_INPUT_CONTROL.in_ToolTip_Size,
								Ist_STRING := 'Password Failed   ',
								Xus_TN_SCREEN := Xus_TN_SCREEN);

			Gst_SysLog_Command := CONCAT('LOGON: ',FB_TN_SC_WRITE_C.Ist_STRING);

		END_IF;
	END_IF;
END_IF;

(* Initialisierung der Daten und Strukturen *)
IF (Xus_TN_SCREEN.in_Page_Number = INT#10 ) THEN
	Xus_TN_SCREEN.in_Page_Number := INT#11;

	(* Clear-Screen (Farbe setzen + Display löschen) *)
	Xus_TN_SCREEN.by_Clear_Screen_Attr := BYTE#16#00;
	Xus_TN_SCREEN.bo_Clear_Screen := TRUE;

	(* Screen initialisieren (mit Leerzeichen füllen) *)
	FB_TN_SC_FILL(	Iin_X1 := INT#00,
					Iin_Y1 := INT#00,
					Iin_X2 := INT#79,
					Iin_Y2 := INT#23,
					Iby_CHAR := BYTE#179,
					Iby_Attr := BYTE#16#76,
					Xus_TN_SCREEN := Xus_TN_SCREEN);

